LIN {X 0.083,Y -526.031,Z 1290.638,A 0.000,B 0.000,C 90.000,E1 330.745} C_DIS
LIN {X 0.274,Y -522.669,Z 1290.634,A 0.000,B 0.000,C 90.000,E1 329.999} C_DIS
LIN {X 0.174,Y -519.078,Z 1290.630,A 0.000,B 0.000,C 90.000,E1 329.282} C_DIS
LIN {X -0.136,Y -515.219,Z 1290.625,A 0.000,B 0.000,C 90.000,E1 328.584} C_DIS
LIN {X 0.084,Y -506.189,Z 1290.616,A 0.000,B 0.000,C 90.000,E1 326.786} C_DIS
LIN {X -0.322,Y -502.917,Z 1290.611,A 0.000,B 0.000,C 90.000,E1 326.087} C_DIS
LIN {X 0.061,Y -500.954,Z 1290.608,A 0.000,B 0.000,C 90.000,E1 325.468} C_DIS
LIN {X -0.178,Y -499.307,Z 1290.605,A 0.000,B 0.000,C 90.000,E1 324.895} C_DIS
LIN {X -0.148,Y -497.632,Z 1290.600,A 0.000,B 0.000,C 90.000,E1 323.989} C_DIS
LIN {X 0.154,Y -496.578,Z 1290.595,A 0.000,B 0.000,C 90.000,E1 323.050} C_DIS
LIN {X 0.309,Y -495.797,Z 1290.588,A 0.000,B 0.000,C 90.000,E1 321.823} C_DIS
LIN {X -0.218,Y -495.460,Z 1290.578,A 0.000,B 0.000,C 90.000,E1 320.070} C_DIS
LIN {X -0.116,Y -495.714,Z 1290.568,A 0.000,B 0.000,C 90.000,E1 318.243} C_DIS
LIN {X -0.048,Y -495.867,Z 1290.561,A 0.000,B 0.000,C 90.000,E1 317.025} C_DIS
LIN {X 0.028,Y -496.080,Z 1290.551,A 0.000,B 0.000,C 90.000,E1 315.202} C_DIS
LIN {X 0.109,Y -496.318,Z 1290.541,A 0.000,B 0.000,C 90.000,E1 313.380} C_DIS
LIN {X -0.001,Y -496.479,Z 1290.536,A 0.000,B 0.000,C 90.000,E1 312.486} C_DIS
LIN {X -0.140,Y -496.309,Z 1290.531,A 0.000,B 0.000,C 90.000,E1 311.595} C_DIS
LIN {X -0.099,Y -495.936,Z 1290.528,A 0.000,B 0.000,C 90.000,E1 310.987} C_DIS
LIN {X -0.062,Y -495.305,Z 1290.524,A 0.000,B 0.000,C 90.000,E1 310.378} C_DIS
LIN {X -0.031,Y -494.227,Z 1290.521,A 0.000,B 0.000,C 90.000,E1 309.769} C_DIS
LIN {X -0.175,Y -493.450,Z 1290.519,A 0.000,B 0.000,C 90.000,E1 309.483} C_DIS
LIN {X 0.062,Y -492.278,Z 1290.518,A 0.000,B 0.000,C 90.000,E1 309.152} C_DIS
LIN {X 0.225,Y -490.280,Z 1290.516,A 0.000,B 0.000,C 90.000,E1 308.830} C_DIS
LIN {X 0.189,Y -473.095,Z 1290.501,A 0.000,B 0.000,C 90.000,E1 306.217} C_DIS
LIN {X -0.156,Y -457.653,Z 1290.486,A 0.000,B 0.000,C 90.000,E1 303.579} C_DIS
LIN {X 0.164,Y -443.847,Z 1290.471,A 0.000,B 0.000,C 90.000,E1 300.797} C_DIS
LIN {X 0.057,Y -430.915,Z 1290.455,A 0.000,B 0.000,C 90.000,E1 297.847} C_DIS
LIN {X -0.181,Y -420.207,Z 1290.439,A 0.000,B 0.000,C 90.000,E1 295.027} C_DIS
LIN {X -0.114,Y -410.389,Z 1290.422,A 0.000,B 0.000,C 90.000,E1 291.950} C_DIS
LIN {X 0.091,Y -403.056,Z 1290.407,A 0.000,B 0.000,C 90.000,E1 289.214} C_DIS
LIN {X 0.053,Y -403.058,Z 1290.407,A 0.000,B 0.000,C 90.000,E1 289.214} C_DIS
LIN {X -0.122,Y -404.702,Z 1290.395,A 0.000,B 0.000,C 90.000,E1 287.094} C_DIS
LIN {X -0.130,Y -406.128,Z 1290.364,A 0.000,B 0.000,C 90.000,E1 281.535} C_DIS
LIN {X -0.087,Y -405.724,Z 1290.356,A 0.000,B 0.000,C 90.000,E1 280.141} C_DIS
LIN {X -0.037,Y -405.688,Z 1290.333,A 0.000,B 0.000,C 90.000,E1 275.967} C_DIS
LIN {X 0.000,Y -403.466,Z 1290.304,A 0.000,B 0.000,C 90.000,E1 270.745} C_DIS
LIN {X -0.032,Y -403.253,Z 1290.302,A 0.000,B 0.000,C 90.000,E1 270.401} C_DIS
LIN {X 0.147,Y -398.874,Z 1290.271,A 0.000,B 0.000,C 90.000,E1 264.780} C_DIS
LIN {X 0.045,Y -393.348,Z 1290.244,A 0.000,B 0.000,C 90.000,E1 259.859} C_DIS
LIN {X -0.033,Y -392.777,Z 1290.240,A 0.000,B 0.000,C 90.000,E1 259.162} C_DIS
LIN {X 0.116,Y -390.126,Z 1290.230,A 0.000,B 0.000,C 90.000,E1 257.465} C_DIS
LIN {X 0.079,Y -390.127,Z 1290.230,A 0.000,B 0.000,C 90.000,E1 257.465} C_DIS
LIN {X -0.160,Y -397.492,Z 1290.208,A 0.000,B 0.000,C 90.000,E1 253.504} C_DIS
LIN {X -0.205,Y -405.860,Z 1290.189,A 0.000,B 0.000,C 90.000,E1 250.007} C_DIS
LIN {X 0.003,Y -414.932,Z 1290.172,A 0.000,B 0.000,C 90.000,E1 246.869} C_DIS
LIN {X 0.012,Y -426.168,Z 1290.154,A 0.000,B 0.000,C 90.000,E1 243.640} C_DIS
LIN {X -0.200,Y -438.462,Z 1290.137,A 0.000,B 0.000,C 90.000,E1 240.667} C_DIS
LIN {X -0.039,Y -451.639,Z 1290.121,A 0.000,B 0.000,C 90.000,E1 237.867} C_DIS
LIN {X 0.118,Y -455.806,Z 1290.117,A 0.000,B 0.000,C 90.000,E1 237.041} C_DIS
LIN {X -0.149,Y -456.438,Z 1290.116,A 0.000,B 0.000,C 90.000,E1 236.914} C_DIS
LIN {X -0.045,Y -457.275,Z 1290.114,A 0.000,B 0.000,C 90.000,E1 236.580} C_DIS
LIN {X 0.059,Y -457.846,Z 1290.113,A 0.000,B 0.000,C 90.000,E1 236.246} C_DIS
LIN {X 0.155,Y -458.486,Z 1290.109,A 0.000,B 0.000,C 90.000,E1 235.595} C_DIS
LIN {X -0.001,Y -458.776,Z 1290.105,A 0.000,B 0.000,C 90.000,E1 234.975} C_DIS
LIN {X 0.222,Y -458.863,Z 1290.100,A 0.000,B 0.000,C 90.000,E1 233.989} C_DIS
LIN {X 0.076,Y -458.567,Z 1290.095,A 0.000,B 0.000,C 90.000,E1 233.050} C_DIS
LIN {X -0.223,Y -457.721,Z 1290.084,A 0.000,B 0.000,C 90.000,E1 231.170} C_DIS
LIN {X 0.129,Y -456.793,Z 1290.070,A 0.000,B 0.000,C 90.000,E1 228.566} C_DIS
LIN {X -0.042,Y -456.332,Z 1290.061,A 0.000,B 0.000,C 90.000,E1 226.986} C_DIS
LIN {X -0.130,Y -455.866,Z 1290.047,A 0.000,B 0.000,C 90.000,E1 224.433} C_DIS
LIN {X -0.137,Y -456.231,Z 1290.027,A 0.000,B 0.000,C 90.000,E1 220.906} C_DIS
LIN {X -0.095,Y -457.345,Z 1290.013,A 0.000,B 0.000,C 90.000,E1 218.338} C_DIS
LIN {X 0.015,Y -461.089,Z 1289.985,A 0.000,B 0.000,C 90.000,E1 213.214} C_DIS
LIN {X -0.103,Y -463.575,Z 1289.972,A 0.000,B 0.000,C 90.000,E1 211.003} C_DIS
LIN {X -0.167,Y -467.366,Z 1289.955,A 0.000,B 0.000,C 90.000,E1 207.847} C_DIS
LIN {X 0.254,Y -470.340,Z 1289.942,A 0.000,B 0.000,C 90.000,E1 205.591} C_DIS
LIN {X -0.201,Y -472.677,Z 1289.934,A 0.000,B 0.000,C 90.000,E1 204.079} C_DIS
LIN {X 0.177,Y -476.348,Z 1289.920,A 0.000,B 0.000,C 90.000,E1 201.535} C_DIS
LIN {X -0.111,Y -479.825,Z 1289.908,A 0.000,B 0.000,C 90.000,E1 199.396} C_DIS
LIN {X 0.138,Y -482.883,Z 1289.897,A 0.000,B 0.000,C 90.000,E1 197.511} C_DIS
LIN {X 0.160,Y -485.987,Z 1289.887,A 0.000,B 0.000,C 90.000,E1 195.662} C_DIS
LIN {X 0.129,Y -489.110,Z 1289.877,A 0.000,B 0.000,C 90.000,E1 193.828} C_DIS
LIN {X 0.160,Y -491.727,Z 1289.869,A 0.000,B 0.000,C 90.000,E1 192.299} C_DIS
LIN {X -0.049,Y -495.342,Z 1289.857,A 0.000,B 0.000,C 90.000,E1 190.197} C_DIS
LIN {X -0.171,Y -498.512,Z 1289.847,A 0.000,B 0.000,C 90.000,E1 188.398} C_DIS
LIN {X 0.073,Y -500.049,Z 1289.842,A 0.000,B 0.000,C 90.000,E1 187.466} C_DIS
LIN {X -0.082,Y -503.094,Z 1289.832,A 0.000,B 0.000,C 90.000,E1 185.682} C_DIS
LIN {X -0.090,Y -505.461,Z 1289.823,A 0.000,B 0.000,C 90.000,E1 184.188} C_DIS
LIN {X 0.046,Y -507.381,Z 1289.817,A 0.000,B 0.000,C 90.000,E1 182.980} C_DIS
LIN {X 0.080,Y -509.631,Z 1289.808,A 0.000,B 0.000,C 90.000,E1 181.489} C_DIS
LIN {X 0.148,Y -511.671,Z 1289.800,A 0.000,B 0.000,C 90.000,E1 180.000} C_DIS
LIN {X -0.259,Y -513.528,Z 1289.792,A 0.000,B 0.000,C 90.000,E1 178.568} C_DIS
LIN {X -0.036,Y -514.856,Z 1289.785,A 0.000,B 0.000,C 90.000,E1 177.364} C_DIS
LIN {X -0.232,Y -515.732,Z 1289.781,A 0.000,B 0.000,C 90.000,E1 176.502} C_DIS
LIN {X 0.096,Y -516.454,Z 1289.776,A 0.000,B 0.000,C 90.000,E1 175.584} C_DIS
LIN {X -0.110,Y -517.200,Z 1289.769,A 0.000,B 0.000,C 90.000,E1 174.432} C_DIS
LIN {X 0.191,Y -517.807,Z 1289.761,A 0.000,B 0.000,C 90.000,E1 172.932} C_DIS
LIN {X 0.081,Y -517.978,Z 1289.756,A 0.000,B 0.000,C 90.000,E1 172.064} C_DIS
LIN {X -0.037,Y -517.969,Z 1289.750,A 0.000,B 0.000,C 90.000,E1 170.905} C_DIS
LIN {X -0.160,Y -517.604,Z 1289.743,A 0.000,B 0.000,C 90.000,E1 169.746} C_DIS
LIN {X -0.199,Y -516.890,Z 1289.736,A 0.000,B 0.000,C 90.000,E1 168.578} C_DIS
LIN {X -0.237,Y -516.175,Z 1289.732,A 0.000,B 0.000,C 90.000,E1 167.701} C_DIS
LIN {X -0.204,Y -514.467,Z 1289.723,A 0.000,B 0.000,C 90.000,E1 166.228} C_DIS
LIN {X -0.251,Y -513.714,Z 1289.720,A 0.000,B 0.000,C 90.000,E1 165.644} C_DIS
LIN {X -0.142,Y -511.511,Z 1289.712,A 0.000,B 0.000,C 90.000,E1 164.157} C_DIS
LIN {X 0.020,Y -508.537,Z 1289.702,A 0.000,B 0.000,C 90.000,E1 162.362} C_DIS
LIN {X 0.154,Y -506.908,Z 1289.697,A 0.000,B 0.000,C 90.000,E1 161.456} C_DIS
LIN {X 0.147,Y -503.458,Z 1289.682,A 0.000,B 0.000,C 90.000,E1 158.773} C_DIS
LIN {X -0.069,Y -502.868,Z 1289.677,A 0.000,B 0.000,C 90.000,E1 157.901} C_DIS
LIN {X 0.176,Y -502.812,Z 1289.672,A 0.000,B 0.000,C 90.000,E1 156.975} C_DIS
LIN {X 0.257,Y -502.910,Z 1289.671,A 0.000,B 0.000,C 90.000,E1 156.666} C_DIS
LIN {X -0.125,Y -503.191,Z 1289.669,A 0.000,B 0.000,C 90.000,E1 156.410} C_DIS
LIN {X 0.035,Y -504.310,Z 1289.666,A 0.000,B 0.000,C 90.000,E1 155.793} C_DIS
LIN {X -0.259,Y -506.027,Z 1289.662,A 0.000,B 0.000,C 90.000,E1 155.229} C_DIS
LIN {X -0.162,Y -507.409,Z 1289.661,A 0.000,B 0.000,C 90.000,E1 154.921} C_DIS
LIN {X 0.330,Y -508.042,Z 1289.660,A 0.000,B 0.000,C 90.000,E1 154.717} C_DIS
LIN {X 0.020,Y -512.118,Z 1289.656,A 0.000,B 0.000,C 90.000,E1 154.076} C_DIS
LIN {X 0.060,Y -519.658,Z 1289.650,A 0.000,B 0.000,C 90.000,E1 152.999} C_DIS
LIN {X -0.046,Y -526.944,Z 1289.645,A 0.000,B 0.000,C 90.000,E1 152.153} C_DIS
LIN {X -0.094,Y -532.653,Z 1289.641,A 0.000,B 0.000,C 90.000,E1 151.435} C_DIS
LIN {X 0.050,Y -540.691,Z 1289.637,A 0.000,B 0.000,C 90.000,E1 150.589} C_DIS
LIN {X -0.215,Y -549.206,Z 1289.633,A 0.000,B 0.000,C 90.000,E1 149.871} C_DIS
LIN {X -0.326,Y -559.542,Z 1289.628,A 0.000,B 0.000,C 90.000,E1 149.076} C_DIS
LIN {X 0.230,Y -576.226,Z 1289.620,A 0.000,B 0.000,C 90.000,E1 147.582} C_DIS
LIN {X -0.049,Y -580.302,Z 1289.618,A 0.000,B 0.000,C 90.000,E1 147.248} C_DIS
LIN {X -0.255,Y -589.432,Z 1289.613,A 0.000,B 0.000,C 90.000,E1 146.421} C_DIS
LIN {X 0.108,Y -595.843,Z 1289.610,A 0.000,B 0.000,C 90.000,E1 145.754} C_DIS
LIN {X 0.154,Y -601.955,Z 1289.606,A 0.000,B 0.000,C 90.000,E1 145.102} C_DIS
LIN {X 0.039,Y -609.405,Z 1289.601,A 0.000,B 0.000,C 90.000,E1 144.196} C_DIS
LIN {X -0.255,Y -613.214,Z 1289.598,A 0.000,B 0.000,C 90.000,E1 143.703} C_DIS
LIN {X -0.190,Y -617.440,Z 1289.595,A 0.000,B 0.000,C 90.000,E1 143.050} C_DIS
LIN {X -0.084,Y -621.380,Z 1289.591,A 0.000,B 0.000,C 90.000,E1 142.396} C_DIS
LIN {X 0.031,Y -625.965,Z 1289.587,A 0.000,B 0.000,C 90.000,E1 141.618} C_DIS
LIN {X 0.207,Y -629.372,Z 1289.583,A 0.000,B 0.000,C 90.000,E1 140.964} C_DIS
LIN {X -0.056,Y -631.927,Z 1289.580,A 0.000,B 0.000,C 90.000,E1 140.481} C_DIS
LIN {X 0.037,Y -636.667,Z 1289.575,A 0.000,B 0.000,C 90.000,E1 139.461} C_DIS
LIN {X 0.215,Y -639.855,Z 1289.571,A 0.000,B 0.000,C 90.000,E1 138.690} C_DIS
LIN {X -0.165,Y -644.960,Z 1289.564,A 0.000,B 0.000,C 90.000,E1 137.472} C_DIS
LIN {X -0.091,Y -650.633,Z 1289.555,A 0.000,B 0.000,C 90.000,E1 135.972} C_DIS
LIN {X -0.331,Y -655.263,Z 1289.549,A 0.000,B 0.000,C 90.000,E1 134.757} C_DIS
LIN {X 0.006,Y -658.983,Z 1289.543,A 0.000,B 0.000,C 90.000,E1 133.743} C_DIS
LIN {X -0.119,Y -664.500,Z 1289.535,A 0.000,B 0.000,C 90.000,E1 132.285} C_DIS
LIN {X -0.103,Y -668.044,Z 1289.530,A 0.000,B 0.000,C 90.000,E1 131.310} C_DIS
LIN {X -0.033,Y -671.477,Z 1289.524,A 0.000,B 0.000,C 90.000,E1 130.334} C_DIS
LIN {X 0.093,Y -675.495,Z 1289.517,A 0.000,B 0.000,C 90.000,E1 129.116} C_DIS
LIN {X -0.154,Y -679.235,Z 1289.511,A 0.000,B 0.000,C 90.000,E1 127.935} C_DIS
LIN {X 0.191,Y -682.761,Z 1289.504,A 0.000,B 0.000,C 90.000,E1 126.710} C_DIS
LIN {X -0.030,Y -684.097,Z 1289.501,A 0.000,B 0.000,C 90.000,E1 126.251} C_DIS
LIN {X 0.396,Y -687.135,Z 1289.495,A 0.000,B 0.000,C 90.000,E1 125.025} C_DIS
LIN {X 0.080,Y -689.867,Z 1289.488,A 0.000,B 0.000,C 90.000,E1 123.865} C_DIS
LIN {X -0.049,Y -691.316,Z 1289.484,A 0.000,B 0.000,C 90.000,E1 123.166} C_DIS
LIN {X -0.300,Y -693.492,Z 1289.478,A 0.000,B 0.000,C 90.000,E1 122.005} C_DIS
LIN {X -0.035,Y -696.136,Z 1289.469,A 0.000,B 0.000,C 90.000,E1 120.335} C_DIS
LIN {X -0.321,Y -698.144,Z 1289.461,A 0.000,B 0.000,C 90.000,E1 118.949} C_DIS
LIN {X 0.121,Y -699.124,Z 1289.456,A 0.000,B 0.000,C 90.000,E1 117.975} C_DIS
LIN {X -0.049,Y -699.821,Z 1289.450,A 0.000,B 0.000,C 90.000,E1 117.052} C_DIS
LIN {X 0.092,Y -699.981,Z 1289.445,A 0.000,B 0.000,C 90.000,E1 116.104} C_DIS
LIN {X 0.003,Y -699.865,Z 1289.443,A 0.000,B 0.000,C 90.000,E1 115.643} C_DIS
LIN {X 0.243,Y -699.577,Z 1289.440,A 0.000,B 0.000,C 90.000,E1 115.155} C_DIS
LIN {X -0.147,Y -699.127,Z 1289.437,A 0.000,B 0.000,C 90.000,E1 114.719} C_DIS
LIN {X -0.250,Y -698.336,Z 1289.435,A 0.000,B 0.000,C 90.000,E1 114.259} C_DIS
LIN {X -0.009,Y -696.698,Z 1289.432,A 0.000,B 0.000,C 90.000,E1 113.770} C_DIS
LIN {X 0.249,Y -695.719,Z 1289.431,A 0.000,B 0.000,C 90.000,E1 113.515} C_DIS
LIN {X -0.161,Y -692.441,Z 1289.428,A 0.000,B 0.000,C 90.000,E1 113.078} C_DIS
LIN {X -0.041,Y -691.488,Z 1289.427,A 0.000,B 0.000,C 90.000,E1 112.950} C_DIS
LIN {X 0.079,Y -690.067,Z 1289.427,A 0.000,B 0.000,C 90.000,E1 112.823} C_DIS
LIN {X -0.317,Y -683.445,Z 1289.425,A 0.000,B 0.000,C 90.000,E1 112.461} C_DIS
LIN {X 0.136,Y -681.325,Z 1289.424,A 0.000,B 0.000,C 90.000,E1 112.333} C_DIS
LIN {X -0.044,Y -678.247,Z 1289.424,A 0.000,B 0.000,C 90.000,E1 112.259} C_DIS
LIN {X -0.416,Y -671.472,Z 1289.423,A 0.000,B 0.000,C 90.000,E1 112.153} C_DIS
LIN {X 0.035,Y -668.069,Z 1289.423,A 0.000,B 0.000,C 90.000,E1 112.078} C_DIS
LIN {X 0.350,Y -663.498,Z 1289.423,A 0.000,B 0.000,C 90.000,E1 112.025} C_DIS
LIN {X 0.281,Y -643.375,Z 1289.423,A 0.000,B 0.000,C 90.000,E1 112.025} C_DIS
LIN {X -0.170,Y -641.107,Z 1289.422,A 0.000,B 0.000,C 90.000,E1 112.025} C_DIS
LIN {X -0.112,Y -638.394,Z 1289.422,A 0.000,B 0.000,C 90.000,E1 111.950} C_DIS
LIN {X -0.146,Y -638.300,Z 1289.422,A 0.000,B 0.000,C 90.000,E1 111.950} C_DIS
LIN {X -0.141,Y -639.010,Z 1289.421,A 0.000,B 0.000,C 90.000,E1 111.770} C_DIS
LIN {X -0.153,Y -641.523,Z 1289.419,A 0.000,B 0.000,C 90.000,E1 111.354} C_DIS
LIN {X -0.195,Y -647.571,Z 1289.414,A 0.000,B 0.000,C 90.000,E1 110.556} C_DIS
LIN {X -0.090,Y -650.233,Z 1289.412,A 0.000,B 0.000,C 90.000,E1 110.174} C_DIS
LIN {X -0.339,Y -654.176,Z 1289.409,A 0.000,B 0.000,C 90.000,E1 109.577} C_DIS
LIN {X 0.331,Y -658.195,Z 1289.405,A 0.000,B 0.000,C 90.000,E1 108.779} C_DIS
LIN {X 0.201,Y -661.735,Z 1289.400,A 0.000,B 0.000,C 90.000,E1 108.055} C_DIS
LIN {X 0.101,Y -664.869,Z 1289.396,A 0.000,B 0.000,C 90.000,E1 107.330} C_DIS
LIN {X -0.080,Y -666.764,Z 1289.394,A 0.000,B 0.000,C 90.000,E1 106.858} C_DIS
LIN {X -0.136,Y -669.232,Z 1289.390,A 0.000,B 0.000,C 90.000,E1 106.134} C_DIS
LIN {X -0.284,Y -670.626,Z 1289.387,A 0.000,B 0.000,C 90.000,E1 105.662} C_DIS
LIN {X 0.102,Y -672.899,Z 1289.382,A 0.000,B 0.000,C 90.000,E1 104.662} C_DIS
LIN {X -0.015,Y -673.828,Z 1289.379,A 0.000,B 0.000,C 90.000,E1 104.189} C_DIS
LIN {X 0.034,Y -674.563,Z 1289.376,A 0.000,B 0.000,C 90.000,E1 103.703} C_DIS
LIN {X -0.285,Y -675.371,Z 1289.372,A 0.000,B 0.000,C 90.000,E1 103.008} C_DIS
LIN {X 0.271,Y -675.698,Z 1289.370,A 0.000,B 0.000,C 90.000,E1 102.479} C_DIS
LIN {X 0.169,Y -675.845,Z 1289.367,A 0.000,B 0.000,C 90.000,E1 102.007} C_DIS
LIN {X 0.064,Y -675.815,Z 1289.364,A 0.000,B 0.000,C 90.000,E1 101.535} C_DIS
LIN {X -0.227,Y -675.337,Z 1289.360,A 0.000,B 0.000,C 90.000,E1 100.838} C_DIS
LIN {X 0.324,Y -674.842,Z 1289.357,A 0.000,B 0.000,C 90.000,E1 100.310} C_DIS
LIN {X 0.088,Y -674.132,Z 1289.355,A 0.000,B 0.000,C 90.000,E1 99.849} C_DIS
LIN {X -0.038,Y -673.123,Z 1289.352,A 0.000,B 0.000,C 90.000,E1 99.378} C_DIS
LIN {X -0.281,Y -671.788,Z 1289.349,A 0.000,B 0.000,C 90.000,E1 98.916} C_DIS
LIN {X 0.135,Y -670.122,Z 1289.347,A 0.000,B 0.000,C 90.000,E1 98.398} C_DIS
LIN {X 0.056,Y -669.245,Z 1289.345,A 0.000,B 0.000,C 90.000,E1 98.163} C_DIS
LIN {X -0.205,Y -667.130,Z 1289.343,A 0.000,B 0.000,C 90.000,E1 97.701} C_DIS
LIN {X 0.091,Y -664.060,Z 1289.339,A 0.000,B 0.000,C 90.000,E1 97.068} C_DIS
LIN {X -0.220,Y -660.538,Z 1289.336,A 0.000,B 0.000,C 90.000,E1 96.486} C_DIS
LIN {X 0.116,Y -657.365,Z 1289.333,A 0.000,B 0.000,C 90.000,E1 95.967} C_DIS
LIN {X 0.322,Y -652.937,Z 1289.330,A 0.000,B 0.000,C 90.000,E1 95.334} C_DIS
LIN {X -0.101,Y -649.078,Z 1289.327,A 0.000,B 0.000,C 90.000,E1 94.878} C_DIS
LIN {X 0.155,Y -644.861,Z 1289.324,A 0.000,B 0.000,C 90.000,E1 94.359} C_DIS
LIN {X -0.260,Y -639.140,Z 1289.321,A 0.000,B 0.000,C 90.000,E1 93.784} C_DIS
LIN {X -0.147,Y -633.038,Z 1289.318,A 0.000,B 0.000,C 90.000,E1 93.154} C_DIS
LIN {X 0.159,Y -627.876,Z 1289.315,A 0.000,B 0.000,C 90.000,E1 92.636} C_DIS
LIN {X -0.115,Y -622.794,Z 1289.312,A 0.000,B 0.000,C 90.000,E1 92.178} C_DIS
LIN {X 0.306,Y -615.979,Z 1289.309,A 0.000,B 0.000,C 90.000,E1 91.547} C_DIS
LIN {X -0.011,Y -608.410,Z 1289.306,A 0.000,B 0.000,C 90.000,E1 91.031} C_DIS
LIN {X -0.016,Y -602.179,Z 1289.304,A 0.000,B 0.000,C 90.000,E1 90.630} C_DIS
LIN {X -0.280,Y -595.714,Z 1289.302,A 0.000,B 0.000,C 90.000,E1 90.286} C_DIS
LIN {X -0.162,Y -588.834,Z 1289.300,A 0.000,B 0.000,C 90.000,E1 89.943} C_DIS
LIN {X -0.242,Y -579.881,Z 1289.298,A 0.000,B 0.000,C 90.000,E1 89.599} C_DIS
LIN {X 0.177,Y -576.140,Z 1289.297,A 0.000,B 0.000,C 90.000,E1 89.427} C_DIS
LIN {X -0.083,Y -571.959,Z 1289.296,A 0.000,B 0.000,C 90.000,E1 89.255} C_DIS
LIN {X 0.024,Y -569.925,Z 1289.295,A 0.000,B 0.000,C 90.000,E1 89.026} C_DIS
LIN {X -0.014,Y -569.915,Z 1289.295,A 0.000,B 0.000,C 90.000,E1 89.026} C_DIS
LIN {X -0.276,Y -569.540,Z 1289.294,A 0.000,B 0.000,C 90.000,E1 88.854} C_DIS
LIN {X 0.074,Y -569.423,Z 1289.293,A 0.000,B 0.000,C 90.000,E1 88.682} C_DIS
LIN {X -0.027,Y -569.681,Z 1289.289,A 0.000,B 0.000,C 90.000,E1 87.993} C_DIS
LIN {X -0.222,Y -572.279,Z 1289.272,A 0.000,B 0.000,C 90.000,E1 85.008} C_DIS
LIN {X -0.109,Y -574.690,Z 1289.260,A 0.000,B 0.000,C 90.000,E1 82.818} C_DIS
LIN {X 0.014,Y -576.977,Z 1289.250,A 0.000,B 0.000,C 90.000,E1 80.905} C_DIS
LIN {X 0.205,Y -578.245,Z 1289.244,A 0.000,B 0.000,C 90.000,E1 79.803} C_DIS
LIN {X 0.058,Y -579.558,Z 1289.236,A 0.000,B 0.000,C 90.000,E1 78.465} C_DIS
LIN {X 0.043,Y -580.781,Z 1289.229,A 0.000,B 0.000,C 90.000,E1 77.117} C_DIS
LIN {X 0.186,Y -581.899,Z 1289.221,A 0.000,B 0.000,C 90.000,E1 75.755} C_DIS
LIN {X -0.029,Y -582.693,Z 1289.215,A 0.000,B 0.000,C 90.000,E1 74.700} C_DIS
LIN {X 0.076,Y -583.456,Z 1289.209,A 0.000,B 0.000,C 90.000,E1 73.614} C_DIS
LIN {X 0.166,Y -584.861,Z 1289.197,A 0.000,B 0.000,C 90.000,E1 71.456} C_DIS
LIN {X -0.239,Y -585.464,Z 1289.191,A 0.000,B 0.000,C 90.000,E1 70.423} C_DIS
LIN {X 0.195,Y -586.369,Z 1289.182,A 0.000,B 0.000,C 90.000,E1 68.773} C_DIS
LIN {X -0.147,Y -587.681,Z 1289.170,A 0.000,B 0.000,C 90.000,E1 66.666} C_DIS
LIN {X 0.111,Y -588.676,Z 1289.163,A 0.000,B 0.000,C 90.000,E1 65.305} C_DIS
LIN {X -0.128,Y -590.074,Z 1289.153,A 0.000,B 0.000,C 90.000,E1 63.461} C_DIS
LIN {X 0.139,Y -591.214,Z 1289.145,A 0.000,B 0.000,C 90.000,E1 62.103} C_DIS
LIN {X -0.002,Y -593.003,Z 1289.135,A 0.000,B 0.000,C 90.000,E1 60.255} C_DIS
LIN {X -0.100,Y -594.899,Z 1289.125,A 0.000,B 0.000,C 90.000,E1 58.408} C_DIS
LIN {X -0.034,Y -596.868,Z 1289.114,A 0.000,B 0.000,C 90.000,E1 56.548} C_DIS
LIN {X -0.150,Y -598.434,Z 1289.105,A 0.000,B 0.000,C 90.000,E1 54.975} C_DIS
LIN {X 0.092,Y -599.906,Z 1289.097,A 0.000,B 0.000,C 90.000,E1 53.371} C_DIS
LIN {X 0.010,Y -601.454,Z 1289.086,A 0.000,B 0.000,C 90.000,E1 51.537} C_DIS
LIN {X 0.071,Y -602.250,Z 1289.081,A 0.000,B 0.000,C 90.000,E1 50.481} C_DIS
LIN {X -0.243,Y -602.804,Z 1289.075,A 0.000,B 0.000,C 90.000,E1 49.461} C_DIS
LIN {X -0.370,Y -603.418,Z 1289.067,A 0.000,B 0.000,C 90.000,E1 48.162} C_DIS
LIN {X 0.161,Y -603.881,Z 1289.059,A 0.000,B 0.000,C 90.000,E1 46.539} C_DIS
LIN {X 0.022,Y -604.056,Z 1289.051,A 0.000,B 0.000,C 90.000,E1 45.243} C_DIS
LIN {X -0.112,Y -603.975,Z 1289.044,A 0.000,B 0.000,C 90.000,E1 43.947} C_DIS
LIN {X 0.145,Y -603.764,Z 1289.040,A 0.000,B 0.000,C 90.000,E1 43.137} C_DIS
LIN {X 0.026,Y -603.400,Z 1289.032,A 0.000,B 0.000,C 90.000,E1 41.838} C_DIS
LIN {X -0.136,Y -603.069,Z 1289.028,A 0.000,B 0.000,C 90.000,E1 41.067} C_DIS
LIN {X 0.232,Y -602.241,Z 1289.018,A 0.000,B 0.000,C 90.000,E1 39.197} C_DIS
LIN {X -0.331,Y -601.777,Z 1289.014,A 0.000,B 0.000,C 90.000,E1 38.463} C_DIS
LIN {X 0.077,Y -600.553,Z 1289.006,A 0.000,B 0.000,C 90.000,E1 37.111} C_DIS
LIN {X -0.015,Y -599.026,Z 1288.999,A 0.000,B 0.000,C 90.000,E1 35.804} C_DIS
LIN {X 0.102,Y -597.464,Z 1288.993,A 0.000,B 0.000,C 90.000,E1 34.739} C_DIS
LIN {X -0.371,Y -596.093,Z 1288.989,A 0.000,B 0.000,C 90.000,E1 33.992} C_DIS
LIN {X 0.192,Y -593.975,Z 1288.983,A 0.000,B 0.000,C 90.000,E1 32.880} C_DIS
LIN {X 0.191,Y -592.025,Z 1288.978,A 0.000,B 0.000,C 90.000,E1 32.084} C_DIS
LIN {X -0.327,Y -589.854,Z 1288.974,A 0.000,B 0.000,C 90.000,E1 31.337} C_DIS
LIN {X -0.064,Y -587.336,Z 1288.969,A 0.000,B 0.000,C 90.000,E1 30.512} C_DIS
LIN {X -0.300,Y -585.501,Z 1288.967,A 0.000,B 0.000,C 90.000,E1 30.001} C_DIS
LIN {X 0.253,Y -583.423,Z 1288.964,A 0.000,B 0.000,C 90.000,E1 29.411} C_DIS
LIN {X 0.147,Y -579.877,Z 1288.959,A 0.000,B 0.000,C 90.000,E1 28.615} C_DIS
LIN {X -0.275,Y -575.881,Z 1288.955,A 0.000,B 0.000,C 90.000,E1 27.847} C_DIS
LIN {X 0.039,Y -571.531,Z 1288.950,A 0.000,B 0.000,C 90.000,E1 27.001} C_DIS
LIN {X 0.046,Y -566.470,Z 1288.946,A 0.000,B 0.000,C 90.000,E1 26.181} C_DIS
LIN {X -0.070,Y -562.902,Z 1288.943,A 0.000,B 0.000,C 90.000,E1 25.643} C_DIS
LIN {X -0.054,Y -558.124,Z 1288.939,A 0.000,B 0.000,C 90.000,E1 24.951} C_DIS
LIN {X -0.077,Y -553.050,Z 1288.935,A 0.000,B 0.000,C 90.000,E1 24.259} C_DIS
LIN {X -0.027,Y -548.578,Z 1288.932,A 0.000,B 0.000,C 90.000,E1 23.695} C_DIS
LIN {X 0.102,Y -540.186,Z 1288.926,A 0.000,B 0.000,C 90.000,E1 22.695} C_DIS
LIN {X -0.105,Y -533.983,Z 1288.922,A 0.000,B 0.000,C 90.000,E1 22.025} C_DIS
LIN {X -0.029,Y -524.966,Z 1288.917,A 0.000,B 0.000,C 90.000,E1 21.046} C_DIS
LIN {X -0.119,Y -518.287,Z 1288.913,A 0.000,B 0.000,C 90.000,E1 20.355} C_DIS
LIN {X -0.137,Y -508.782,Z 1288.908,A 0.000,B 0.000,C 90.000,E1 19.396} C_DIS
LIN {X -0.208,Y -503.243,Z 1288.905,A 0.000,B 0.000,C 90.000,E1 18.852} C_DIS
LIN {X 0.077,Y -494.971,Z 1288.900,A 0.000,B 0.000,C 90.000,E1 18.000} C_DIS
LIN {X 0.183,Y -484.832,Z 1288.895,A 0.000,B 0.000,C 90.000,E1 17.040} C_DIS
LIN {X -0.018,Y -474.573,Z 1288.890,A 0.000,B 0.000,C 90.000,E1 16.134} C_DIS
LIN {X 0.122,Y -464.230,Z 1288.885,A 0.000,B 0.000,C 90.000,E1 15.190} C_DIS
LIN {X 0.153,Y -445.086,Z 1288.875,A 0.000,B 0.000,C 90.000,E1 13.411} C_DIS
LIN {X -0.172,Y -424.752,Z 1288.863,A 0.000,B 0.000,C 90.000,E1 11.422} C_DIS
LIN {X 0.099,Y -410.388,Z 1288.855,A 0.000,B 0.000,C 90.000,E1 9.849} C_DIS
LIN {X -0.008,Y -400.468,Z 1288.849,A 0.000,B 0.000,C 90.000,E1 8.746} C_DIS
LIN {X -0.102,Y -396.120,Z 1288.845,A 0.000,B 0.000,C 90.000,E1 8.163} C_DIS
LIN {X 0.035,Y -395.163,Z 1288.844,A 0.000,B 0.000,C 90.000,E1 7.936} C_DIS
LIN {X -0.002,Y -395.150,Z 1288.844,A 0.000,B 0.000,C 90.000,E1 7.936} C_DIS
LIN {X -0.040,Y -395.154,Z 1288.844,A 0.000,B 0.000,C 90.000,E1 7.936} C_DIS
LIN {X -0.078,Y -395.167,Z 1288.844,A 0.000,B 0.000,C 90.000,E1 7.936} C_DIS
LIN {X 0.011,Y -396.219,Z 1288.843,A 0.000,B 0.000,C 90.000,E1 7.757} C_DIS
LIN {X 0.107,Y -399.293,Z 1288.842,A 0.000,B 0.000,C 90.000,E1 7.473} C_DIS
LIN {X -0.156,Y -405.364,Z 1288.839,A 0.000,B 0.000,C 90.000,E1 7.125} C_DIS
LIN {X 0.185,Y -410.605,Z 1288.838,A 0.000,B 0.000,C 90.000,E1 6.777} C_DIS
LIN {X 0.170,Y -416.965,Z 1288.836,A 0.000,B 0.000,C 90.000,E1 6.372} C_DIS
LIN {X -0.097,Y -423.351,Z 1288.833,A 0.000,B 0.000,C 90.000,E1 5.967} C_DIS
LIN {X 0.216,Y -431.048,Z 1288.830,A 0.000,B 0.000,C 90.000,E1 5.334} C_DIS
LIN {X 0.134,Y -441.954,Z 1288.825,A 0.000,B 0.000,C 90.000,E1 4.473} C_DIS
LIN {X 0.220,Y -452.449,Z 1288.820,A 0.000,B 0.000,C 90.000,E1 3.555} C_DIS
LIN {X -0.073,Y -459.789,Z 1288.816,A 0.000,B 0.000,C 90.000,E1 2.922} C_DIS
LIN {X -0.038,Y -466.686,Z 1288.813,A 0.000,B 0.000,C 90.000,E1 2.236} C_DIS
LIN {X 0.051,Y -473.467,Z 1288.808,A 0.000,B 0.000,C 90.000,E1 1.489} C_DIS
LIN {X -0.124,Y -479.927,Z 1288.804,A 0.000,B 0.000,C 90.000,E1 0.745} C_DIS
LIN {X -0.178,Y -483.660,Z 1288.802,A 0.000,B 0.000,C 90.000,E1 0.286} C_DIS
LIN {X 0.011,Y -489.433,Z 1288.797,A 0.000,B 0.000,C 90.000,E1 359.484} C_DIS
LIN {X -0.141,Y -494.604,Z 1288.793,A 0.000,B 0.000,C 90.000,E1 358.740} C_DIS
LIN {X -0.051,Y -500.266,Z 1288.788,A 0.000,B 0.000,C 90.000,E1 357.822} C_DIS
LIN {X -0.110,Y -504.696,Z 1288.784,A 0.000,B 0.000,C 90.000,E1 357.078} C_DIS
LIN {X 0.201,Y -508.065,Z 1288.780,A 0.000,B 0.000,C 90.000,E1 356.445} C_DIS
LIN {X 0.245,Y -511.946,Z 1288.776,A 0.000,B 0.000,C 90.000,E1 355.698} C_DIS
LIN {X 0.242,Y -517.047,Z 1288.771,A 0.000,B 0.000,C 90.000,E1 354.666} C_DIS
LIN {X -0.168,Y -521.582,Z 1288.765,A 0.000,B 0.000,C 90.000,E1 353.685} C_DIS
LIN {X 0.055,Y -524.615,Z 1288.761,A 0.000,B 0.000,C 90.000,E1 352.932} C_DIS
LIN {X 0.004,Y -526.826,Z 1288.758,A 0.000,B 0.000,C 90.000,E1 352.356} C_DIS
LIN {X 0.018,Y -530.883,Z 1288.751,A 0.000,B 0.000,C 90.000,E1 351.197} C_DIS
LIN {X 0.046,Y -533.605,Z 1288.746,A 0.000,B 0.000,C 90.000,E1 350.330} C_DIS
LIN {X 0.192,Y -536.124,Z 1288.742,A 0.000,B 0.000,C 90.000,E1 349.454} C_DIS
LIN {X -0.158,Y -538.320,Z 1288.737,A 0.000,B 0.000,C 90.000,E1 348.634} C_DIS
LIN {X 0.044,Y -540.358,Z 1288.732,A 0.000,B 0.000,C 90.000,E1 347.757} C_DIS
LIN {X -0.184,Y -542.773,Z 1288.726,A 0.000,B 0.000,C 90.000,E1 346.645} C_DIS
LIN {X 0.189,Y -544.323,Z 1288.721,A 0.000,B 0.000,C 90.000,E1 345.755} C_DIS
LIN {X -0.085,Y -545.663,Z 1288.716,A 0.000,B 0.000,C 90.000,E1 344.936} C_DIS
LIN {X 0.032,Y -547.070,Z 1288.710,A 0.000,B 0.000,C 90.000,E1 343.795} C_DIS
LIN {X 0.264,Y -548.264,Z 1288.702,A 0.000,B 0.000,C 90.000,E1 342.362} C_DIS
LIN {X 0.165,Y -548.687,Z 1288.698,A 0.000,B 0.000,C 90.000,E1 341.529} C_DIS
LIN {X -0.277,Y -548.795,Z 1288.693,A 0.000,B 0.000,C 90.000,E1 340.732} C_DIS
LIN {X 0.066,Y -548.428,Z 1288.687,A 0.000,B 0.000,C 90.000,E1 339.571} C_DIS
LIN {X -0.119,Y -548.045,Z 1288.683,A 0.000,B 0.000,C 90.000,E1 339.028} C_DIS
LIN {X -0.099,Y -546.792,Z 1288.677,A 0.000,B 0.000,C 90.000,E1 337.901} C_DIS
LIN {X -0.300,Y -545.907,Z 1288.674,A 0.000,B 0.000,C 90.000,E1 337.358} C_DIS
LIN {X 0.195,Y -544.099,Z 1288.668,A 0.000,B 0.000,C 90.000,E1 336.177} C_DIS
LIN {X -0.059,Y -543.358,Z 1288.666,A 0.000,B 0.000,C 90.000,E1 335.921} C_DIS
LIN {X 0.181,Y -542.845,Z 1288.665,A 0.000,B 0.000,C 90.000,E1 335.613} C_DIS
LIN {X 0.125,Y -539.908,Z 1288.658,A 0.000,B 0.000,C 90.000,E1 334.485} C_DIS
LIN {X 0.045,Y -537.391,Z 1288.654,A 0.000,B 0.000,C 90.000,E1 333.640} C_DIS
LIN {X 0.143,Y -533.647,Z 1288.647,A 0.000,B 0.000,C 90.000,E1 332.487} C_DIS
LIN {X 0.296,Y -531.650,Z 1288.644,A 0.000,B 0.000,C 90.000,E1 331.897} C_DIS
LIN {X -0.285,Y -529.516,Z 1288.641,A 0.000,B 0.000,C 90.000,E1 331.385} C_DIS
LIN {X -0.055,Y -526.481,Z 1288.637,A 0.000,B 0.000,C 90.000,E1 330.639} C_DIS
LIN {X 0.020,Y -521.568,Z 1288.631,A 0.000,B 0.000,C 90.000,E1 329.616} C_DIS
LIN {X 0.174,Y -517.769,Z 1288.627,A 0.000,B 0.000,C 90.000,E1 328.869} C_DIS
LIN {X 0.012,Y -508.458,Z 1288.617,A 0.000,B 0.000,C 90.000,E1 327.120} C_DIS
LIN {X -0.058,Y -503.575,Z 1288.612,A 0.000,B 0.000,C 90.000,E1 326.087} C_DIS
LIN {X 0.015,Y -500.604,Z 1288.607,A 0.000,B 0.000,C 90.000,E1 325.182} C_DIS
LIN {X 0.182,Y -499.198,Z 1288.603,A 0.000,B 0.000,C 90.000,E1 324.562} C_DIS
LIN {X -0.198,Y -497.680,Z 1288.598,A 0.000,B 0.000,C 90.000,E1 323.703} C_DIS
LIN {X 0.106,Y -496.795,Z 1288.593,A 0.000,B 0.000,C 90.000,E1 322.763} C_DIS
LIN {X 0.264,Y -496.105,Z 1288.587,A 0.000,B 0.000,C 90.000,E1 321.537} C_DIS
LIN {X -0.118,Y -495.919,Z 1288.578,A 0.000,B 0.000,C 90.000,E1 320.070} C_DIS
LIN {X -0.005,Y -496.149,Z 1288.568,A 0.000,B 0.000,C 90.000,E1 318.243} C_DIS
LIN {X -0.104,Y -496.360,Z 1288.560,A 0.000,B 0.000,C 90.000,E1 316.743} C_DIS
LIN {X -0.006,Y -496.573,Z 1288.550,A 0.000,B 0.000,C 90.000,E1 314.919} C_DIS
LIN {X -0.225,Y -496.987,Z 1288.536,A 0.000,B 0.000,C 90.000,E1 312.528} C_DIS
LIN {X -0.133,Y -497.179,Z 1288.529,A 0.000,B 0.000,C 90.000,E1 311.310} C_DIS
LIN {X 0.100,Y -496.918,Z 1288.524,A 0.000,B 0.000,C 90.000,E1 310.378} C_DIS
LIN {X 0.006,Y -496.164,Z 1288.519,A 0.000,B 0.000,C 90.000,E1 309.483} C_DIS
LIN {X -0.271,Y -495.267,Z 1288.516,A 0.000,B 0.000,C 90.000,E1 308.910} C_DIS
LIN {X -0.100,Y -494.647,Z 1288.514,A 0.000,B 0.000,C 90.000,E1 308.588} C_DIS
LIN {X 0.147,Y -493.807,Z 1288.513,A 0.000,B 0.000,C 90.000,E1 308.257} C_DIS
LIN {X 0.228,Y -493.242,Z 1288.512,A 0.000,B 0.000,C 90.000,E1 308.096} C_DIS
LIN {X 0.006,Y -492.494,Z 1288.511,A 0.000,B 0.000,C 90.000,E1 307.971} C_DIS
LIN {X -0.187,Y -474.919,Z 1288.496,A 0.000,B 0.000,C 90.000,E1 305.231} C_DIS
LIN {X -0.079,Y -460.039,Z 1288.481,A 0.000,B 0.000,C 90.000,E1 302.546} C_DIS
LIN {X -0.182,Y -446.015,Z 1288.465,A 0.000,B 0.000,C 90.000,E1 299.667} C_DIS
LIN {X -0.019,Y -433.673,Z 1288.448,A 0.000,B 0.000,C 90.000,E1 296.693} C_DIS
LIN {X 0.016,Y -422.378,Z 1288.431,A 0.000,B 0.000,C 90.000,E1 293.515} C_DIS
LIN {X -0.017,Y -412.304,Z 1288.412,A 0.000,B 0.000,C 90.000,E1 290.120} C_DIS
LIN {X -0.181,Y -404.756,Z 1288.395,A 0.000,B 0.000,C 90.000,E1 287.040} C_DIS
LIN {X -0.219,Y -404.745,Z 1288.395,A 0.000,B 0.000,C 90.000,E1 287.040} C_DIS
LIN {X -0.174,Y -406.154,Z 1288.364,A 0.000,B 0.000,C 90.000,E1 281.478} C_DIS
LIN {X -0.075,Y -405.681,Z 1288.333,A 0.000,B 0.000,C 90.000,E1 275.910} C_DIS
LIN {X -0.004,Y -403.567,Z 1288.306,A 0.000,B 0.000,C 90.000,E1 271.031} C_DIS
LIN {X -0.069,Y -403.188,Z 1288.302,A 0.000,B 0.000,C 90.000,E1 270.344} C_DIS
LIN {X 0.165,Y -399.069,Z 1288.273,A 0.000,B 0.000,C 90.000,E1 265.065} C_DIS
LIN {X 0.105,Y -398.785,Z 1288.271,A 0.000,B 0.000,C 90.000,E1 264.723} C_DIS
LIN {X -0.133,Y -393.373,Z 1288.244,A 0.000,B 0.000,C 90.000,E1 259.916} C_DIS
LIN {X 0.215,Y -393.371,Z 1288.244,A 0.000,B 0.000,C 90.000,E1 259.859} C_DIS
LIN {X -0.047,Y -400.123,Z 1288.220,A 0.000,B 0.000,C 90.000,E1 255.574} C_DIS
LIN {X -0.231,Y -408.324,Z 1288.199,A 0.000,B 0.000,C 90.000,E1 251.764} C_DIS
LIN {X 0.067,Y -417.618,Z 1288.179,A 0.000,B 0.000,C 90.000,E1 248.284} C_DIS
LIN {X -0.183,Y -428.146,Z 1288.162,A 0.000,B 0.000,C 90.000,E1 245.101} C_DIS
LIN {X -0.145,Y -439.718,Z 1288.145,A 0.000,B 0.000,C 90.000,E1 242.103} C_DIS
LIN {X 0.180,Y -452.936,Z 1288.129,A 0.000,B 0.000,C 90.000,E1 239.125} C_DIS
LIN {X 0.111,Y -456.914,Z 1288.124,A 0.000,B 0.000,C 90.000,E1 238.329} C_DIS
LIN {X 0.219,Y -458.091,Z 1288.122,A 0.000,B 0.000,C 90.000,E1 237.995} C_DIS
LIN {X -0.058,Y -458.768,Z 1288.121,A 0.000,B 0.000,C 90.000,E1 237.709} C_DIS
LIN {X 0.175,Y -459.535,Z 1288.117,A 0.000,B 0.000,C 90.000,E1 237.041} C_DIS
LIN {X 0.029,Y -459.957,Z 1288.114,A 0.000,B 0.000,C 90.000,E1 236.421} C_DIS
LIN {X -0.114,Y -460.117,Z 1288.110,A 0.000,B 0.000,C 90.000,E1 235.801} C_DIS
LIN {X 0.127,Y -459.954,Z 1288.105,A 0.000,B 0.000,C 90.000,E1 234.815} C_DIS
LIN {X 0.107,Y -459.392,Z 1288.098,A 0.000,B 0.000,C 90.000,E1 233.543} C_DIS
LIN {X -0.074,Y -458.348,Z 1288.085,A 0.000,B 0.000,C 90.000,E1 231.331} C_DIS
LIN {X -0.050,Y -457.412,Z 1288.071,A 0.000,B 0.000,C 90.000,E1 228.771} C_DIS
LIN {X -0.121,Y -456.766,Z 1288.058,A 0.000,B 0.000,C 90.000,E1 226.539} C_DIS
LIN {X 0.173,Y -456.335,Z 1288.041,A 0.000,B 0.000,C 90.000,E1 223.299} C_DIS
LIN {X -0.077,Y -457.117,Z 1288.021,A 0.000,B 0.000,C 90.000,E1 219.806} C_DIS
LIN {X -0.113,Y -457.987,Z 1288.010,A 0.000,B 0.000,C 90.000,E1 217.890} C_DIS
LIN {X 0.018,Y -462.599,Z 1287.979,A 0.000,B 0.000,C 90.000,E1 212.133} C_DIS
LIN {X 0.062,Y -464.415,Z 1287.970,A 0.000,B 0.000,C 90.000,E1 210.541} C_DIS
LIN {X -0.196,Y -467.072,Z 1287.958,A 0.000,B 0.000,C 90.000,E1 208.359} C_DIS
LIN {X 0.216,Y -469.988,Z 1287.945,A 0.000,B 0.000,C 90.000,E1 206.104} C_DIS
LIN {X -0.131,Y -473.184,Z 1287.933,A 0.000,B 0.000,C 90.000,E1 203.951} C_DIS
LIN {X -0.182,Y -476.875,Z 1287.919,A 0.000,B 0.000,C 90.000,E1 201.461} C_DIS
LIN {X -0.003,Y -479.865,Z 1287.909,A 0.000,B 0.000,C 90.000,E1 199.577} C_DIS
LIN {X 0.248,Y -482.968,Z 1287.899,A 0.000,B 0.000,C 90.000,E1 197.692} C_DIS
LIN {X -0.193,Y -486.113,Z 1287.888,A 0.000,B 0.000,C 90.000,E1 195.898} C_DIS
LIN {X -0.106,Y -488.233,Z 1287.881,A 0.000,B 0.000,C 90.000,E1 194.662} C_DIS
LIN {X 0.025,Y -490.871,Z 1287.873,A 0.000,B 0.000,C 90.000,E1 193.119} C_DIS
LIN {X 0.085,Y -492.982,Z 1287.866,A 0.000,B 0.000,C 90.000,E1 191.895} C_DIS
LIN {X 0.182,Y -495.627,Z 1287.858,A 0.000,B 0.000,C 90.000,E1 190.366} C_DIS
LIN {X 0.062,Y -498.844,Z 1287.848,A 0.000,B 0.000,C 90.000,E1 188.568} C_DIS
LIN {X 0.241,Y -500.472,Z 1287.843,A 0.000,B 0.000,C 90.000,E1 187.644} C_DIS
LIN {X 0.157,Y -503.549,Z 1287.833,A 0.000,B 0.000,C 90.000,E1 185.853} C_DIS
LIN {X 0.154,Y -505.985,Z 1287.824,A 0.000,B 0.000,C 90.000,E1 184.359} C_DIS
LIN {X -0.237,Y -507.991,Z 1287.818,A 0.000,B 0.000,C 90.000,E1 183.212} C_DIS
LIN {X -0.165,Y -510.308,Z 1287.809,A 0.000,B 0.000,C 90.000,E1 181.718} C_DIS
LIN {X -0.004,Y -512.007,Z 1287.803,A 0.000,B 0.000,C 90.000,E1 180.516} C_DIS
LIN {X -0.247,Y -513.289,Z 1287.798,A 0.000,B 0.000,C 90.000,E1 179.656} C_DIS
LIN {X -0.098,Y -515.208,Z 1287.790,A 0.000,B 0.000,C 90.000,E1 178.165} C_DIS
LIN {X 0.132,Y -516.543,Z 1287.783,A 0.000,B 0.000,C 90.000,E1 176.963} C_DIS
LIN {X -0.082,Y -517.687,Z 1287.777,A 0.000,B 0.000,C 90.000,E1 175.812} C_DIS
LIN {X 0.178,Y -518.705,Z 1287.769,A 0.000,B 0.000,C 90.000,E1 174.318} C_DIS
LIN {X 0.002,Y -519.303,Z 1287.762,A 0.000,B 0.000,C 90.000,E1 173.166} C_DIS
LIN {X -0.103,Y -519.613,Z 1287.756,A 0.000,B 0.000,C 90.000,E1 172.008} C_DIS
LIN {X -0.199,Y -519.756,Z 1287.749,A 0.000,B 0.000,C 90.000,E1 170.849} C_DIS
LIN {X 0.217,Y -519.550,Z 1287.744,A 0.000,B 0.000,C 90.000,E1 169.926} C_DIS
LIN {X 0.201,Y -519.045,Z 1287.738,A 0.000,B 0.000,C 90.000,E1 168.757} C_DIS
LIN {X 0.177,Y -518.279,Z 1287.731,A 0.000,B 0.000,C 90.000,E1 167.589} C_DIS
LIN {X 0.267,Y -517.406,Z 1287.726,A 0.000,B 0.000,C 90.000,E1 166.700} C_DIS
LIN {X -0.181,Y -515.769,Z 1287.718,A 0.000,B 0.000,C 90.000,E1 165.283} C_DIS
LIN {X -0.060,Y -513.438,Z 1287.708,A 0.000,B 0.000,C 90.000,E1 163.504} C_DIS
LIN {X 0.082,Y -511.677,Z 1287.702,A 0.000,B 0.000,C 90.000,E1 162.308} C_DIS
LIN {X -0.187,Y -509.660,Z 1287.694,A 0.000,B 0.000,C 90.000,E1 160.859} C_DIS
LIN {X -0.217,Y -508.050,Z 1287.684,A 0.000,B 0.000,C 90.000,E1 159.082} C_DIS
LIN {X 0.088,Y -507.644,Z 1287.679,A 0.000,B 0.000,C 90.000,E1 158.156} C_DIS
LIN {X -0.082,Y -507.875,Z 1287.674,A 0.000,B 0.000,C 90.000,E1 157.283} C_DIS
LIN {X 0.118,Y -508.359,Z 1287.671,A 0.000,B 0.000,C 90.000,E1 156.666} C_DIS
LIN {X -0.146,Y -509.257,Z 1287.667,A 0.000,B 0.000,C 90.000,E1 156.102} C_DIS
LIN {X 0.059,Y -510.468,Z 1287.664,A 0.000,B 0.000,C 90.000,E1 155.485} C_DIS
LIN {X -0.196,Y -512.710,Z 1287.661,A 0.000,B 0.000,C 90.000,E1 154.921} C_DIS
LIN {X 0.310,Y -513.608,Z 1287.660,A 0.000,B 0.000,C 90.000,E1 154.717} C_DIS
LIN {X 0.251,Y -515.631,Z 1287.657,A 0.000,B 0.000,C 90.000,E1 154.280} C_DIS
LIN {X -0.159,Y -522.656,Z 1287.651,A 0.000,B 0.000,C 90.000,E1 153.256} C_DIS
LIN {X 0.014,Y -527.329,Z 1287.648,A 0.000,B 0.000,C 90.000,E1 152.666} C_DIS
LIN {X 0.195,Y -529.511,Z 1287.647,A 0.000,B 0.000,C 90.000,E1 152.410} C_DIS
LIN {X 0.037,Y -536.879,Z 1287.642,A 0.000,B 0.000,C 90.000,E1 151.591} C_DIS
LIN {X 0.264,Y -543.431,Z 1287.639,A 0.000,B 0.000,C 90.000,E1 150.923} C_DIS
LIN {X -0.169,Y -547.634,Z 1287.637,A 0.000,B 0.000,C 90.000,E1 150.589} C_DIS
LIN {X -0.207,Y -550.541,Z 1287.635,A 0.000,B 0.000,C 90.000,E1 150.333} C_DIS
LIN {X -0.049,Y -555.841,Z 1287.633,A 0.000,B 0.000,C 90.000,E1 149.871} C_DIS
LIN {X -0.186,Y -562.846,Z 1287.629,A 0.000,B 0.000,C 90.000,E1 149.282} C_DIS
LIN {X 0.105,Y -575.235,Z 1287.623,A 0.000,B 0.000,C 90.000,E1 148.152} C_DIS
LIN {X -0.278,Y -583.311,Z 1287.619,A 0.000,B 0.000,C 90.000,E1 147.454} C_DIS
LIN {X 0.133,Y -589.782,Z 1287.616,A 0.000,B 0.000,C 90.000,E1 146.786} C_DIS
LIN {X -0.042,Y -594.851,Z 1287.613,A 0.000,B 0.000,C 90.000,E1 146.294} C_DIS
LIN {X 0.139,Y -599.657,Z 1287.610,A 0.000,B 0.000,C 90.000,E1 145.754} C_DIS
LIN {X 0.004,Y -603.033,Z 1287.608,A 0.000,B 0.000,C 90.000,E1 145.388} C_DIS
LIN {X 0.167,Y -607.235,Z 1287.605,A 0.000,B 0.000,C 90.000,E1 144.848} C_DIS
LIN {X -0.141,Y -611.242,Z 1287.602,A 0.000,B 0.000,C 90.000,E1 144.356} C_DIS
LIN {X -0.390,Y -614.058,Z 1287.600,A 0.000,B 0.000,C 90.000,E1 143.989} C_DIS
LIN {X 0.175,Y -618.286,Z 1287.596,A 0.000,B 0.000,C 90.000,E1 143.290} C_DIS
LIN {X -0.208,Y -622.205,Z 1287.593,A 0.000,B 0.000,C 90.000,E1 142.683} C_DIS
LIN {X -0.084,Y -626.540,Z 1287.588,A 0.000,B 0.000,C 90.000,E1 141.904} C_DIS
LIN {X 0.077,Y -630.573,Z 1287.584,A 0.000,B 0.000,C 90.000,E1 141.126} C_DIS
LIN {X -0.200,Y -633.642,Z 1287.581,A 0.000,B 0.000,C 90.000,E1 140.517} C_DIS
LIN {X 0.318,Y -638.213,Z 1287.575,A 0.000,B 0.000,C 90.000,E1 139.461} C_DIS
LIN {X 0.088,Y -641.293,Z 1287.571,A 0.000,B 0.000,C 90.000,E1 138.728} C_DIS
LIN {X 0.230,Y -645.212,Z 1287.565,A 0.000,B 0.000,C 90.000,E1 137.715} C_DIS
LIN {X -0.104,Y -649.838,Z 1287.558,A 0.000,B 0.000,C 90.000,E1 136.500} C_DIS
LIN {X 0.073,Y -655.267,Z 1287.550,A 0.000,B 0.000,C 90.000,E1 135.000} C_DIS
LIN {X -0.142,Y -661.516,Z 1287.541,A 0.000,B 0.000,C 90.000,E1 133.299} C_DIS
LIN {X -0.181,Y -666.002,Z 1287.534,A 0.000,B 0.000,C 90.000,E1 132.081} C_DIS
LIN {X -0.137,Y -670.234,Z 1287.527,A 0.000,B 0.000,C 90.000,E1 130.862} C_DIS
LIN {X -0.028,Y -674.269,Z 1287.520,A 0.000,B 0.000,C 90.000,E1 129.644} C_DIS
LIN {X 0.117,Y -677.343,Z 1287.515,A 0.000,B 0.000,C 90.000,E1 128.669} C_DIS
LIN {X -0.124,Y -680.256,Z 1287.510,A 0.000,B 0.000,C 90.000,E1 127.729} C_DIS
LIN {X 0.241,Y -683.689,Z 1287.503,A 0.000,B 0.000,C 90.000,E1 126.503} C_DIS
LIN {X 0.258,Y -686.723,Z 1287.496,A 0.000,B 0.000,C 90.000,E1 125.311} C_DIS
LIN {X -0.268,Y -689.014,Z 1287.491,A 0.000,B 0.000,C 90.000,E1 124.405} C_DIS
LIN {X 0.188,Y -691.128,Z 1287.486,A 0.000,B 0.000,C 90.000,E1 123.420} C_DIS
LIN {X 0.159,Y -693.753,Z 1287.478,A 0.000,B 0.000,C 90.000,E1 122.005} C_DIS
LIN {X 0.182,Y -696.038,Z 1287.470,A 0.000,B 0.000,C 90.000,E1 120.590} C_DIS
LIN {X 0.334,Y -697.124,Z 1287.466,A 0.000,B 0.000,C 90.000,E1 119.873} C_DIS
LIN {X -0.197,Y -698.724,Z 1287.460,A 0.000,B 0.000,C 90.000,E1 118.743} C_DIS
LIN {X -0.019,Y -699.476,Z 1287.456,A 0.000,B 0.000,C 90.000,E1 118.025} C_DIS
LIN {X 0.116,Y -700.223,Z 1287.451,A 0.000,B 0.000,C 90.000,E1 117.078} C_DIS
LIN {X -0.047,Y -700.397,Z 1287.445,A 0.000,B 0.000,C 90.000,E1 116.155} C_DIS
LIN {X -0.083,Y -700.420,Z 1287.444,A 0.000,B 0.000,C 90.000,E1 115.924} C_DIS
LIN {X 0.102,Y -700.045,Z 1287.440,A 0.000,B 0.000,C 90.000,E1 115.207} C_DIS
LIN {X -0.287,Y -699.623,Z 1287.438,A 0.000,B 0.000,C 90.000,E1 114.771} C_DIS
LIN {X 0.248,Y -698.850,Z 1287.435,A 0.000,B 0.000,C 90.000,E1 114.259} C_DIS
LIN {X 0.228,Y -698.208,Z 1287.434,A 0.000,B 0.000,C 90.000,E1 114.027} C_DIS
LIN {X 0.114,Y -696.446,Z 1287.431,A 0.000,B 0.000,C 90.000,E1 113.567} C_DIS
LIN {X -0.036,Y -695.748,Z 1287.430,A 0.000,B 0.000,C 90.000,E1 113.462} C_DIS
LIN {X -0.174,Y -692.349,Z 1287.428,A 0.000,B 0.000,C 90.000,E1 113.003} C_DIS
LIN {X -0.321,Y -691.177,Z 1287.427,A 0.000,B 0.000,C 90.000,E1 112.898} C_DIS
LIN {X -0.200,Y -689.354,Z 1287.427,A 0.000,B 0.000,C 90.000,E1 112.770} C_DIS
LIN {X -0.081,Y -687.123,Z 1287.426,A 0.000,B 0.000,C 90.000,E1 112.642} C_DIS
LIN {X 0.041,Y -683.361,Z 1287.425,A 0.000,B 0.000,C 90.000,E1 112.408} C_DIS
LIN {X -0.134,Y -681.095,Z 1287.424,A 0.000,B 0.000,C 90.000,E1 112.333} C_DIS
LIN {X -0.286,Y -678.946,Z 1287.424,A 0.000,B 0.000,C 90.000,E1 112.280} C_DIS
LIN {X 0.058,Y -670.940,Z 1287.423,A 0.000,B 0.000,C 90.000,E1 112.099} C_DIS
LIN {X -0.234,Y -663.585,Z 1287.423,A 0.000,B 0.000,C 90.000,E1 112.078} C_DIS
LIN {X 0.326,Y -642.480,Z 1287.423,A 0.000,B 0.000,C 90.000,E1 112.025} C_DIS
LIN {X 0.210,Y -639.088,Z 1287.422,A 0.000,B 0.000,C 90.000,E1 111.972} C_DIS
LIN {X -0.208,Y -637.906,Z 1287.422,A 0.000,B 0.000,C 90.000,E1 111.972} C_DIS
LIN {X -0.011,Y -637.823,Z 1287.422,A 0.000,B 0.000,C 90.000,E1 111.950} C_DIS
LIN {X 0.156,Y -638.311,Z 1287.421,A 0.000,B 0.000,C 90.000,E1 111.791} C_DIS
LIN {X 0.180,Y -638.945,Z 1287.421,A 0.000,B 0.000,C 90.000,E1 111.663} C_DIS
LIN {X 0.202,Y -641.377,Z 1287.418,A 0.000,B 0.000,C 90.000,E1 111.280} C_DIS
LIN {X -0.089,Y -647.007,Z 1287.414,A 0.000,B 0.000,C 90.000,E1 110.556} C_DIS
LIN {X 0.014,Y -649.703,Z 1287.412,A 0.000,B 0.000,C 90.000,E1 110.174} C_DIS
LIN {X -0.197,Y -654.347,Z 1287.408,A 0.000,B 0.000,C 90.000,E1 109.450} C_DIS
LIN {X -0.196,Y -657.677,Z 1287.405,A 0.000,B 0.000,C 90.000,E1 108.833} C_DIS
LIN {X 0.291,Y -661.205,Z 1287.401,A 0.000,B 0.000,C 90.000,E1 108.055} C_DIS
LIN {X 0.187,Y -664.386,Z 1287.396,A 0.000,B 0.000,C 90.000,E1 107.330} C_DIS
LIN {X 0.003,Y -666.307,Z 1287.394,A 0.000,B 0.000,C 90.000,E1 106.858} C_DIS
LIN {X -0.057,Y -668.795,Z 1287.390,A 0.000,B 0.000,C 90.000,E1 106.134} C_DIS
LIN {X -0.209,Y -670.241,Z 1287.387,A 0.000,B 0.000,C 90.000,E1 105.662} C_DIS
LIN {X 0.173,Y -672.511,Z 1287.382,A 0.000,B 0.000,C 90.000,E1 104.662} C_DIS
LIN {X 0.054,Y -673.466,Z 1287.379,A 0.000,B 0.000,C 90.000,E1 104.189} C_DIS
LIN {X 0.100,Y -674.230,Z 1287.376,A 0.000,B 0.000,C 90.000,E1 103.703} C_DIS
LIN {X -0.223,Y -675.008,Z 1287.372,A 0.000,B 0.000,C 90.000,E1 103.008} C_DIS
LIN {X -0.328,Y -675.362,Z 1287.370,A 0.000,B 0.000,C 90.000,E1 102.535} C_DIS
LIN {X 0.228,Y -675.508,Z 1287.367,A 0.000,B 0.000,C 90.000,E1 102.007} C_DIS
LIN {X 0.121,Y -675.477,Z 1287.364,A 0.000,B 0.000,C 90.000,E1 101.535} C_DIS
LIN {X -0.173,Y -674.968,Z 1287.360,A 0.000,B 0.000,C 90.000,E1 100.838} C_DIS
LIN {X -0.288,Y -674.471,Z 1287.358,A 0.000,B 0.000,C 90.000,E1 100.366} C_DIS
LIN {X 0.137,Y -673.728,Z 1287.355,A 0.000,B 0.000,C 90.000,E1 99.849} C_DIS
LIN {X 0.008,Y -672.751,Z 1287.352,A 0.000,B 0.000,C 90.000,E1 99.378} C_DIS
LIN {X -0.237,Y -671.414,Z 1287.349,A 0.000,B 0.000,C 90.000,E1 98.916} C_DIS
LIN {X 0.176,Y -669.739,Z 1287.347,A 0.000,B 0.000,C 90.000,E1 98.398} C_DIS
LIN {X 0.096,Y -668.836,Z 1287.345,A 0.000,B 0.000,C 90.000,E1 98.163} C_DIS
LIN {X -0.168,Y -666.721,Z 1287.343,A 0.000,B 0.000,C 90.000,E1 97.701} C_DIS
LIN {X 0.124,Y -663.649,Z 1287.339,A 0.000,B 0.000,C 90.000,E1 97.068} C_DIS
LIN {X -0.191,Y -660.109,Z 1287.336,A 0.000,B 0.000,C 90.000,E1 96.486} C_DIS
LIN {X 0.142,Y -656.886,Z 1287.333,A 0.000,B 0.000,C 90.000,E1 95.967} C_DIS
LIN {X 0.344,Y -652.411,Z 1287.330,A 0.000,B 0.000,C 90.000,E1 95.334} C_DIS
LIN {X -0.082,Y -648.526,Z 1287.327,A 0.000,B 0.000,C 90.000,E1 94.878} C_DIS
LIN {X 0.170,Y -644.245,Z 1287.324,A 0.000,B 0.000,C 90.000,E1 94.359} C_DIS
LIN {X 0.266,Y -638.376,Z 1287.321,A 0.000,B 0.000,C 90.000,E1 93.726} C_DIS
LIN {X -0.152,Y -633.491,Z 1287.318,A 0.000,B 0.000,C 90.000,E1 93.269} C_DIS
LIN {X 0.190,Y -628.344,Z 1287.315,A 0.000,B 0.000,C 90.000,E1 92.751} C_DIS
LIN {X 0.251,Y -622.151,Z 1287.312,A 0.000,B 0.000,C 90.000,E1 92.178} C_DIS
LIN {X 0.287,Y -615.431,Z 1287.309,A 0.000,B 0.000,C 90.000,E1 91.604} C_DIS
LIN {X -0.092,Y -609.468,Z 1287.307,A 0.000,B 0.000,C 90.000,E1 91.203} C_DIS
LIN {X -0.242,Y -603.182,Z 1287.304,A 0.000,B 0.000,C 90.000,E1 90.802} C_DIS
LIN {X 0.281,Y -595.102,Z 1287.302,A 0.000,B 0.000,C 90.000,E1 90.286} C_DIS
LIN {X 0.039,Y -589.975,Z 1287.300,A 0.000,B 0.000,C 90.000,E1 90.057} C_DIS
LIN {X -0.054,Y -582.828,Z 1287.299,A 0.000,B 0.000,C 90.000,E1 89.771} C_DIS
LIN {X 0.157,Y -575.815,Z 1287.297,A 0.000,B 0.000,C 90.000,E1 89.484} C_DIS
LIN {X 0.190,Y -572.195,Z 1287.296,A 0.000,B 0.000,C 90.000,E1 89.312} C_DIS
LIN {X 0.141,Y -572.097,Z 1287.296,A 0.000,B 0.000,C 90.000,E1 89.312} C_DIS
LIN {X 0.239,Y -569.807,Z 1287.295,A 0.000,B 0.000,C 90.000,E1 89.026} C_DIS
LIN {X 0.197,Y -569.781,Z 1287.295,A 0.000,B 0.000,C 90.000,E1 89.026} C_DIS
LIN {X -0.047,Y -569.409,Z 1287.294,A 0.000,B 0.000,C 90.000,E1 88.854} C_DIS
LIN {X -0.074,Y -569.368,Z 1287.292,A 0.000,B 0.000,C 90.000,E1 88.568} C_DIS
LIN {X 0.126,Y -572.483,Z 1287.271,A 0.000,B 0.000,C 90.000,E1 84.723} C_DIS
LIN {X 0.234,Y -574.908,Z 1287.259,A 0.000,B 0.000,C 90.000,E1 82.534} C_DIS
LIN {X -0.218,Y -577.189,Z 1287.248,A 0.000,B 0.000,C 90.000,E1 80.679} C_DIS
LIN {X 0.073,Y -578.395,Z 1287.242,A 0.000,B 0.000,C 90.000,E1 79.567} C_DIS
LIN {X -0.071,Y -579.668,Z 1287.235,A 0.000,B 0.000,C 90.000,E1 78.229} C_DIS
LIN {X 0.259,Y -580.651,Z 1287.229,A 0.000,B 0.000,C 90.000,E1 77.117} C_DIS
LIN {X -0.164,Y -581.771,Z 1287.221,A 0.000,B 0.000,C 90.000,E1 75.811} C_DIS
LIN {X 0.183,Y -582.569,Z 1287.215,A 0.000,B 0.000,C 90.000,E1 74.700} C_DIS
LIN {X -0.047,Y -583.467,Z 1287.208,A 0.000,B 0.000,C 90.000,E1 73.378} C_DIS
LIN {X 0.039,Y -584.928,Z 1287.196,A 0.000,B 0.000,C 90.000,E1 71.221} C_DIS
LIN {X -0.019,Y -586.054,Z 1287.184,A 0.000,B 0.000,C 90.000,E1 69.082} C_DIS
LIN {X 0.171,Y -587.356,Z 1287.172,A 0.000,B 0.000,C 90.000,E1 66.922} C_DIS
LIN {X -0.227,Y -588.521,Z 1287.163,A 0.000,B 0.000,C 90.000,E1 65.357} C_DIS
LIN {X 0.173,Y -589.740,Z 1287.154,A 0.000,B 0.000,C 90.000,E1 63.717} C_DIS
LIN {X -0.192,Y -591.091,Z 1287.145,A 0.000,B 0.000,C 90.000,E1 62.153} C_DIS
LIN {X 0.186,Y -592.882,Z 1287.135,A 0.000,B 0.000,C 90.000,E1 60.255} C_DIS
LIN {X 0.086,Y -594.778,Z 1287.125,A 0.000,B 0.000,C 90.000,E1 58.408} C_DIS
LIN {X 0.151,Y -596.746,Z 1287.114,A 0.000,B 0.000,C 90.000,E1 56.548} C_DIS
LIN {X 0.031,Y -598.297,Z 1287.105,A 0.000,B 0.000,C 90.000,E1 54.975} C_DIS
LIN {X -0.210,Y -599.768,Z 1287.097,A 0.000,B 0.000,C 90.000,E1 53.417} C_DIS
LIN {X -0.060,Y -601.112,Z 1287.088,A 0.000,B 0.000,C 90.000,E1 51.823} C_DIS
LIN {X -0.137,Y -602.103,Z 1287.081,A 0.000,B 0.000,C 90.000,E1 50.517} C_DIS
LIN {X 0.177,Y -602.792,Z 1287.073,A 0.000,B 0.000,C 90.000,E1 49.175} C_DIS
LIN {X 0.045,Y -603.373,Z 1287.066,A 0.000,B 0.000,C 90.000,E1 47.877} C_DIS
LIN {X -0.109,Y -603.756,Z 1287.059,A 0.000,B 0.000,C 90.000,E1 46.581} C_DIS
LIN {X -0.036,Y -603.925,Z 1287.053,A 0.000,B 0.000,C 90.000,E1 45.526} C_DIS
LIN {X 0.251,Y -603.890,Z 1287.046,A 0.000,B 0.000,C 90.000,E1 44.190} C_DIS
LIN {X 0.093,Y -603.750,Z 1287.041,A 0.000,B 0.000,C 90.000,E1 43.419} C_DIS
LIN {X 0.188,Y -603.295,Z 1287.033,A 0.000,B 0.000,C 90.000,E1 41.838} C_DIS
LIN {X 0.025,Y -602.964,Z 1287.028,A 0.000,B 0.000,C 90.000,E1 41.067} C_DIS
LIN {X 0.389,Y -602.137,Z 1287.018,A 0.000,B 0.000,C 90.000,E1 39.197} C_DIS
LIN {X -0.175,Y -601.675,Z 1287.014,A 0.000,B 0.000,C 90.000,E1 38.463} C_DIS
LIN {X -0.247,Y -600.446,Z 1287.006,A 0.000,B 0.000,C 90.000,E1 37.156} C_DIS
LIN {X 0.137,Y -598.904,Z 1286.999,A 0.000,B 0.000,C 90.000,E1 35.804} C_DIS
LIN {X 0.018,Y -597.771,Z 1286.995,A 0.000,B 0.000,C 90.000,E1 35.025} C_DIS
LIN {X -0.115,Y -596.494,Z 1286.990,A 0.000,B 0.000,C 90.000,E1 34.246} C_DIS
LIN {X 0.122,Y -594.457,Z 1286.984,A 0.000,B 0.000,C 90.000,E1 33.166} C_DIS
LIN {X -0.374,Y -592.631,Z 1286.980,A 0.000,B 0.000,C 90.000,E1 32.418} C_DIS
LIN {X -0.072,Y -590.501,Z 1286.976,A 0.000,B 0.000,C 90.000,E1 31.592} C_DIS
LIN {X 0.009,Y -588.949,Z 1286.973,A 0.000,B 0.000,C 90.000,E1 31.052} C_DIS
LIN {X -0.039,Y -586.304,Z 1286.968,A 0.000,B 0.000,C 90.000,E1 30.256} C_DIS
LIN {X -0.279,Y -584.382,Z 1286.965,A 0.000,B 0.000,C 90.000,E1 29.745} C_DIS
LIN {X -0.242,Y -582.212,Z 1286.962,A 0.000,B 0.000,C 90.000,E1 29.205} C_DIS
LIN {X 0.216,Y -579.139,Z 1286.958,A 0.000,B 0.000,C 90.000,E1 28.487} C_DIS
LIN {X -0.213,Y -575.090,Z 1286.954,A 0.000,B 0.000,C 90.000,E1 27.719} C_DIS
LIN {X 0.173,Y -571.449,Z 1286.950,A 0.000,B 0.000,C 90.000,E1 27.001} C_DIS
LIN {X 0.178,Y -566.385,Z 1286.946,A 0.000,B 0.000,C 90.000,E1 26.181} C_DIS
LIN {X -0.091,Y -563.711,Z 1286.943,A 0.000,B 0.000,C 90.000,E1 25.796} C_DIS
LIN {X 0.177,Y -558.990,Z 1286.939,A 0.000,B 0.000,C 90.000,E1 25.079} C_DIS
LIN {X 0.050,Y -552.952,Z 1286.935,A 0.000,B 0.000,C 90.000,E1 24.259} C_DIS
LIN {X 0.098,Y -548.474,Z 1286.932,A 0.000,B 0.000,C 90.000,E1 23.695} C_DIS
LIN {X 0.015,Y -540.088,Z 1286.926,A 0.000,B 0.000,C 90.000,E1 22.717} C_DIS
LIN {X -0.015,Y -533.820,Z 1286.922,A 0.000,B 0.000,C 90.000,E1 22.025} C_DIS
LIN {X -0.036,Y -524.711,Z 1286.917,A 0.000,B 0.000,C 90.000,E1 21.046} C_DIS
LIN {X -0.127,Y -518.024,Z 1286.913,A 0.000,B 0.000,C 90.000,E1 20.355} C_DIS
LIN {X -0.259,Y -507.129,Z 1286.907,A 0.000,B 0.000,C 90.000,E1 19.268} C_DIS
LIN {X 0.074,Y -494.684,Z 1286.900,A 0.000,B 0.000,C 90.000,E1 18.000} C_DIS
LIN {X -0.165,Y -486.021,Z 1286.896,A 0.000,B 0.000,C 90.000,E1 17.221} C_DIS
LIN {X 0.104,Y -475.812,Z 1286.891,A 0.000,B 0.000,C 90.000,E1 16.260} C_DIS
LIN {X 0.192,Y -463.954,Z 1286.885,A 0.000,B 0.000,C 90.000,E1 15.190} C_DIS
LIN {X 0.244,Y -444.863,Z 1286.875,A 0.000,B 0.000,C 90.000,E1 13.411} C_DIS
LIN {X -0.107,Y -421.712,Z 1286.862,A 0.000,B 0.000,C 90.000,E1 11.130} C_DIS
LIN {X 0.169,Y -400.374,Z 1286.849,A 0.000,B 0.000,C 90.000,E1 8.746} C_DIS
LIN {X 0.055,Y -396.009,Z 1286.845,A 0.000,B 0.000,C 90.000,E1 8.163} C_DIS
LIN {X -0.005,Y -395.181,Z 1286.844,A 0.000,B 0.000,C 90.000,E1 7.992} C_DIS
LIN {X -0.043,Y -395.159,Z 1286.844,A 0.000,B 0.000,C 90.000,E1 7.992} C_DIS
LIN {X 0.044,Y -395.199,Z 1286.844,A 0.000,B 0.000,C 90.000,E1 7.936} C_DIS
LIN {X 0.006,Y -395.216,Z 1286.844,A 0.000,B 0.000,C 90.000,E1 7.936} C_DIS
LIN {X 0.170,Y -396.173,Z 1286.843,A 0.000,B 0.000,C 90.000,E1 7.757} C_DIS
LIN {X -0.128,Y -399.243,Z 1286.842,A 0.000,B 0.000,C 90.000,E1 7.530} C_DIS
LIN {X -0.074,Y -403.575,Z 1286.840,A 0.000,B 0.000,C 90.000,E1 7.239} C_DIS
LIN {X -0.025,Y -410.511,Z 1286.838,A 0.000,B 0.000,C 90.000,E1 6.834} C_DIS
LIN {X -0.040,Y -416.873,Z 1286.836,A 0.000,B 0.000,C 90.000,E1 6.429} C_DIS
LIN {X 0.082,Y -423.251,Z 1286.833,A 0.000,B 0.000,C 90.000,E1 5.967} C_DIS
LIN {X -0.022,Y -430.944,Z 1286.830,A 0.000,B 0.000,C 90.000,E1 5.391} C_DIS
LIN {X 0.032,Y -441.672,Z 1286.825,A 0.000,B 0.000,C 90.000,E1 4.531} C_DIS
LIN {X 0.183,Y -452.171,Z 1286.820,A 0.000,B 0.000,C 90.000,E1 3.612} C_DIS
LIN {X -0.070,Y -459.506,Z 1286.817,A 0.000,B 0.000,C 90.000,E1 2.980} C_DIS
LIN {X -0.041,Y -466.472,Z 1286.813,A 0.000,B 0.000,C 90.000,E1 2.293} C_DIS
LIN {X 0.062,Y -473.294,Z 1286.809,A 0.000,B 0.000,C 90.000,E1 1.547} C_DIS
LIN {X -0.218,Y -479.510,Z 1286.805,A 0.000,B 0.000,C 90.000,E1 0.859} C_DIS
LIN {X -0.091,Y -484.435,Z 1286.801,A 0.000,B 0.000,C 90.000,E1 0.229} C_DIS
LIN {X 0.013,Y -489.872,Z 1286.797,A 0.000,B 0.000,C 90.000,E1 359.484} C_DIS
LIN {X -0.136,Y -495.044,Z 1286.793,A 0.000,B 0.000,C 90.000,E1 358.740} C_DIS
LIN {X -0.040,Y -500.739,Z 1286.788,A 0.000,B 0.000,C 90.000,E1 357.822} C_DIS
LIN {X -0.095,Y -505.201,Z 1286.784,A 0.000,B 0.000,C 90.000,E1 357.078} C_DIS
LIN {X -0.084,Y -509.376,Z 1286.780,A 0.000,B 0.000,C 90.000,E1 356.331} C_DIS
LIN {X -0.033,Y -513.223,Z 1286.776,A 0.000,B 0.000,C 90.000,E1 355.584} C_DIS
LIN {X 0.027,Y -518.293,Z 1286.770,A 0.000,B 0.000,C 90.000,E1 354.546} C_DIS
LIN {X 0.097,Y -522.738,Z 1286.764,A 0.000,B 0.000,C 90.000,E1 353.514} C_DIS
LIN {X 0.041,Y -526.331,Z 1286.759,A 0.000,B 0.000,C 90.000,E1 352.648} C_DIS
LIN {X 0.044,Y -530.469,Z 1286.753,A 0.000,B 0.000,C 90.000,E1 351.489} C_DIS
LIN {X 0.066,Y -533.339,Z 1286.748,A 0.000,B 0.000,C 90.000,E1 350.622} C_DIS
LIN {X 0.207,Y -535.904,Z 1286.743,A 0.000,B 0.000,C 90.000,E1 349.746} C_DIS
LIN {X -0.146,Y -538.196,Z 1286.738,A 0.000,B 0.000,C 90.000,E1 348.926} C_DIS
LIN {X 0.128,Y -540.947,Z 1286.732,A 0.000,B 0.000,C 90.000,E1 347.757} C_DIS
LIN {X -0.091,Y -543.361,Z 1286.726,A 0.000,B 0.000,C 90.000,E1 346.645} C_DIS
LIN {X 0.072,Y -544.474,Z 1286.723,A 0.000,B 0.000,C 90.000,E1 346.061} C_DIS
LIN {X 0.022,Y -546.334,Z 1286.716,A 0.000,B 0.000,C 90.000,E1 344.936} C_DIS
LIN {X 0.147,Y -547.737,Z 1286.710,A 0.000,B 0.000,C 90.000,E1 343.795} C_DIS
LIN {X 0.052,Y -548.492,Z 1286.705,A 0.000,B 0.000,C 90.000,E1 342.960} C_DIS
LIN {X -0.042,Y -549.173,Z 1286.701,A 0.000,B 0.000,C 90.000,E1 342.127} C_DIS
LIN {X 0.041,Y -549.537,Z 1286.696,A 0.000,B 0.000,C 90.000,E1 341.275} C_DIS
LIN {X -0.133,Y -549.600,Z 1286.693,A 0.000,B 0.000,C 90.000,E1 340.732} C_DIS
LIN {X -0.042,Y -549.377,Z 1286.688,A 0.000,B 0.000,C 90.000,E1 339.880} C_DIS
LIN {X -0.221,Y -549.132,Z 1286.685,A 0.000,B 0.000,C 90.000,E1 339.337} C_DIS
LIN {X 0.059,Y -548.341,Z 1286.680,A 0.000,B 0.000,C 90.000,E1 338.465} C_DIS
LIN {X 0.128,Y -547.304,Z 1286.676,A 0.000,B 0.000,C 90.000,E1 337.614} C_DIS
LIN {X -0.110,Y -544.979,Z 1286.668,A 0.000,B 0.000,C 90.000,E1 336.230} C_DIS
LIN {X -0.114,Y -543.906,Z 1286.665,A 0.000,B 0.000,C 90.000,E1 335.665} C_DIS
LIN {X 0.128,Y -543.271,Z 1286.663,A 0.000,B 0.000,C 90.000,E1 335.357} C_DIS
LIN {X -0.127,Y -542.376,Z 1286.662,A 0.000,B 0.000,C 90.000,E1 335.101} C_DIS
LIN {X -0.107,Y -541.056,Z 1286.659,A 0.000,B 0.000,C 90.000,E1 334.537} C_DIS
LIN {X -0.170,Y -538.591,Z 1286.654,A 0.000,B 0.000,C 90.000,E1 333.691} C_DIS
LIN {X -0.048,Y -534.826,Z 1286.647,A 0.000,B 0.000,C 90.000,E1 332.538} C_DIS
LIN {X 0.012,Y -530.608,Z 1286.641,A 0.000,B 0.000,C 90.000,E1 331.385} C_DIS
LIN {X -0.008,Y -527.621,Z 1286.637,A 0.000,B 0.000,C 90.000,E1 330.667} C_DIS
LIN {X -0.115,Y -522.605,Z 1286.631,A 0.000,B 0.000,C 90.000,E1 329.665} C_DIS
LIN {X -0.049,Y -519.581,Z 1286.628,A 0.000,B 0.000,C 90.000,E1 329.076} C_DIS
LIN {X 0.257,Y -507.846,Z 1286.616,A 0.000,B 0.000,C 90.000,E1 326.834} C_DIS
LIN {X -0.134,Y -504.344,Z 1286.612,A 0.000,B 0.000,C 90.000,E1 326.135} C_DIS
LIN {X -0.222,Y -501.237,Z 1286.607,A 0.000,B 0.000,C 90.000,E1 325.261} C_DIS
LIN {X 0.240,Y -499.788,Z 1286.604,A 0.000,B 0.000,C 90.000,E1 324.609} C_DIS
LIN {X 0.272,Y -498.212,Z 1286.599,A 0.000,B 0.000,C 90.000,E1 323.703} C_DIS
LIN {X 0.015,Y -497.481,Z 1286.595,A 0.000,B 0.000,C 90.000,E1 323.130} C_DIS
LIN {X 0.183,Y -496.687,Z 1286.589,A 0.000,B 0.000,C 90.000,E1 321.904} C_DIS
LIN {X -0.188,Y -496.306,Z 1286.580,A 0.000,B 0.000,C 90.000,E1 320.436} C_DIS
LIN {X -0.063,Y -496.548,Z 1286.570,A 0.000,B 0.000,C 90.000,E1 318.609} C_DIS
LIN {X 0.063,Y -496.806,Z 1286.560,A 0.000,B 0.000,C 90.000,E1 316.782} C_DIS
LIN {X -0.192,Y -497.032,Z 1286.550,A 0.000,B 0.000,C 90.000,E1 315.000} C_DIS
LIN {X 0.306,Y -497.430,Z 1286.536,A 0.000,B 0.000,C 90.000,E1 312.528} C_DIS
LIN {X -0.107,Y -497.757,Z 1286.528,A 0.000,B 0.000,C 90.000,E1 311.067} C_DIS
LIN {X -0.056,Y -497.842,Z 1286.525,A 0.000,B 0.000,C 90.000,E1 310.458} C_DIS
LIN {X -0.140,Y -497.644,Z 1286.520,A 0.000,B 0.000,C 90.000,E1 309.564} C_DIS
LIN {X 0.161,Y -497.038,Z 1286.515,A 0.000,B 0.000,C 90.000,E1 308.624} C_DIS
LIN {X 0.202,Y -496.334,Z 1286.511,A 0.000,B 0.000,C 90.000,E1 308.016} C_DIS
LIN {X 0.066,Y -495.853,Z 1286.510,A 0.000,B 0.000,C 90.000,E1 307.729} C_DIS
LIN {X -0.069,Y -495.241,Z 1286.508,A 0.000,B 0.000,C 90.000,E1 307.443} C_DIS
LIN {X -0.207,Y -494.392,Z 1286.506,A 0.000,B 0.000,C 90.000,E1 307.156} C_DIS
LIN {X -0.127,Y -493.836,Z 1286.505,A 0.000,B 0.000,C 90.000,E1 306.996} C_DIS
LIN {X 0.050,Y -493.107,Z 1286.505,A 0.000,B 0.000,C 90.000,E1 306.824} C_DIS
LIN {X -0.005,Y -476.240,Z 1286.489,A 0.000,B 0.000,C 90.000,E1 304.072} C_DIS
LIN {X -0.100,Y -461.185,Z 1286.474,A 0.000,B 0.000,C 90.000,E1 301.258} C_DIS
LIN {X 0.004,Y -447.852,Z 1286.458,A 0.000,B 0.000,C 90.000,E1 298.359} C_DIS
LIN {X 0.036,Y -436.149,Z 1286.441,A 0.000,B 0.000,C 90.000,E1 295.412} C_DIS
LIN {X 0.121,Y -426.000,Z 1286.425,A 0.000,B 0.000,C 90.000,E1 292.408} C_DIS
LIN {X 0.097,Y -416.449,Z 1286.406,A 0.000,B 0.000,C 90.000,E1 289.033} C_DIS
LIN {X 0.208,Y -407.944,Z 1286.385,A 0.000,B 0.000,C 90.000,E1 285.245} C_DIS
LIN {X -0.125,Y -405.115,Z 1286.376,A 0.000,B 0.000,C 90.000,E1 283.772} C_DIS
LIN {X -0.163,Y -405.116,Z 1286.376,A 0.000,B 0.000,C 90.000,E1 283.772} C_DIS
LIN {X -0.136,Y -406.152,Z 1286.364,A 0.000,B 0.000,C 90.000,E1 281.478} C_DIS
LIN {X -0.038,Y -405.682,Z 1286.333,A 0.000,B 0.000,C 90.000,E1 275.910} C_DIS
LIN {X 0.034,Y -403.568,Z 1286.306,A 0.000,B 0.000,C 90.000,E1 271.031} C_DIS
LIN {X -0.031,Y -403.194,Z 1286.302,A 0.000,B 0.000,C 90.000,E1 270.344} C_DIS
LIN {X 0.201,Y -399.072,Z 1286.273,A 0.000,B 0.000,C 90.000,E1 265.065} C_DIS
LIN {X 0.143,Y -398.792,Z 1286.271,A 0.000,B 0.000,C 90.000,E1 264.723} C_DIS
LIN {X 0.110,Y -396.575,Z 1286.262,A 0.000,B 0.000,C 90.000,E1 263.053} C_DIS
LIN {X 0.071,Y -396.573,Z 1286.261,A 0.000,B 0.000,C 90.000,E1 263.053} C_DIS
LIN {X 0.144,Y -402.593,Z 1286.234,A 0.000,B 0.000,C 90.000,E1 258.049} C_DIS
LIN {X -0.141,Y -410.228,Z 1286.211,A 0.000,B 0.000,C 90.000,E1 253.921} C_DIS
LIN {X -0.048,Y -418.451,Z 1286.192,A 0.000,B 0.000,C 90.000,E1 250.477} C_DIS
LIN {X -0.102,Y -428.442,Z 1286.173,A 0.000,B 0.000,C 90.000,E1 247.102} C_DIS
LIN {X -0.139,Y -439.651,Z 1286.155,A 0.000,B 0.000,C 90.000,E1 243.948} C_DIS
LIN {X -0.076,Y -451.888,Z 1286.139,A 0.000,B 0.000,C 90.000,E1 241.001} C_DIS
LIN {X 0.048,Y -458.614,Z 1286.131,A 0.000,B 0.000,C 90.000,E1 239.537} C_DIS
LIN {X 0.163,Y -459.612,Z 1286.129,A 0.000,B 0.000,C 90.000,E1 239.203} C_DIS
LIN {X -0.113,Y -460.209,Z 1286.127,A 0.000,B 0.000,C 90.000,E1 238.918} C_DIS
LIN {X -0.106,Y -460.910,Z 1286.124,A 0.000,B 0.000,C 90.000,E1 238.280} C_DIS
LIN {X -0.247,Y -461.253,Z 1286.120,A 0.000,B 0.000,C 90.000,E1 237.661} C_DIS
LIN {X -0.254,Y -461.332,Z 1286.115,A 0.000,B 0.000,C 90.000,E1 236.707} C_DIS
LIN {X 0.253,Y -461.261,Z 1286.111,A 0.000,B 0.000,C 90.000,E1 236.008} C_DIS
LIN {X -0.015,Y -460.574,Z 1286.104,A 0.000,B 0.000,C 90.000,E1 234.769} C_DIS
LIN {X -0.165,Y -459.446,Z 1286.092,A 0.000,B 0.000,C 90.000,E1 232.557} C_DIS
LIN {X -0.159,Y -458.596,Z 1286.081,A 0.000,B 0.000,C 90.000,E1 230.642} C_DIS
LIN {X 0.121,Y -457.934,Z 1286.071,A 0.000,B 0.000,C 90.000,E1 228.690} C_DIS
LIN {X 0.065,Y -457.271,Z 1286.058,A 0.000,B 0.000,C 90.000,E1 226.458} C_DIS
LIN {X 0.035,Y -456.832,Z 1286.042,A 0.000,B 0.000,C 90.000,E1 223.581} C_DIS
LIN {X -0.225,Y -457.518,Z 1286.023,A 0.000,B 0.000,C 90.000,E1 220.092} C_DIS
LIN {X 0.121,Y -458.393,Z 1286.010,A 0.000,B 0.000,C 90.000,E1 217.810} C_DIS
LIN {X 0.026,Y -462.999,Z 1285.978,A 0.000,B 0.000,C 90.000,E1 212.084} C_DIS
LIN {X -0.082,Y -464.831,Z 1285.969,A 0.000,B 0.000,C 90.000,E1 210.512} C_DIS
LIN {X 0.114,Y -465.994,Z 1285.964,A 0.000,B 0.000,C 90.000,E1 209.539} C_DIS
LIN {X 0.235,Y -469.106,Z 1285.950,A 0.000,B 0.000,C 90.000,E1 207.001} C_DIS
LIN {X 0.068,Y -472.162,Z 1285.938,A 0.000,B 0.000,C 90.000,E1 204.823} C_DIS
LIN {X 0.073,Y -474.499,Z 1285.929,A 0.000,B 0.000,C 90.000,E1 203.259} C_DIS
LIN {X -0.118,Y -478.323,Z 1285.916,A 0.000,B 0.000,C 90.000,E1 200.791} C_DIS
LIN {X 0.090,Y -481.843,Z 1285.903,A 0.000,B 0.000,C 90.000,E1 198.598} C_DIS
LIN {X 0.231,Y -485.045,Z 1285.893,A 0.000,B 0.000,C 90.000,E1 196.732} C_DIS
LIN {X 0.176,Y -488.265,Z 1285.883,A 0.000,B 0.000,C 90.000,E1 194.898} C_DIS
LIN {X -0.167,Y -490.930,Z 1285.874,A 0.000,B 0.000,C 90.000,E1 193.411} C_DIS
LIN {X -0.109,Y -493.607,Z 1285.866,A 0.000,B 0.000,C 90.000,E1 191.883} C_DIS
LIN {X -0.101,Y -496.306,Z 1285.858,A 0.000,B 0.000,C 90.000,E1 190.366} C_DIS
LIN {X -0.208,Y -499.591,Z 1285.848,A 0.000,B 0.000,C 90.000,E1 188.568} C_DIS
LIN {X -0.099,Y -501.750,Z 1285.841,A 0.000,B 0.000,C 90.000,E1 187.352} C_DIS
LIN {X -0.089,Y -504.389,Z 1285.833,A 0.000,B 0.000,C 90.000,E1 185.853} C_DIS
LIN {X -0.077,Y -506.885,Z 1285.824,A 0.000,B 0.000,C 90.000,E1 184.359} C_DIS
LIN {X 0.052,Y -508.935,Z 1285.818,A 0.000,B 0.000,C 90.000,E1 183.154} C_DIS
LIN {X 0.143,Y -511.318,Z 1285.809,A 0.000,B 0.000,C 90.000,E1 181.661} C_DIS
LIN {X 0.165,Y -513.994,Z 1285.800,A 0.000,B 0.000,C 90.000,E1 179.885} C_DIS
LIN {X 0.261,Y -516.382,Z 1285.790,A 0.000,B 0.000,C 90.000,E1 178.108} C_DIS
LIN {X -0.008,Y -517.797,Z 1285.783,A 0.000,B 0.000,C 90.000,E1 176.963} C_DIS
LIN {X -0.203,Y -519.015,Z 1285.777,A 0.000,B 0.000,C 90.000,E1 175.812} C_DIS
LIN {X 0.082,Y -520.149,Z 1285.769,A 0.000,B 0.000,C 90.000,E1 174.318} C_DIS
LIN {X -0.074,Y -520.840,Z 1285.762,A 0.000,B 0.000,C 90.000,E1 173.166} C_DIS
LIN {X -0.231,Y -521.369,Z 1285.754,A 0.000,B 0.000,C 90.000,E1 171.724} C_DIS
LIN {X -0.228,Y -521.510,Z 1285.749,A 0.000,B 0.000,C 90.000,E1 170.849} C_DIS
LIN {X 0.211,Y -521.335,Z 1285.743,A 0.000,B 0.000,C 90.000,E1 169.634} C_DIS
LIN {X 0.220,Y -521.079,Z 1285.738,A 0.000,B 0.000,C 90.000,E1 168.757} C_DIS
LIN {X -0.282,Y -520.195,Z 1285.730,A 0.000,B 0.000,C 90.000,E1 167.353} C_DIS
LIN {X -0.173,Y -519.128,Z 1285.723,A 0.000,B 0.000,C 90.000,E1 166.172} C_DIS
LIN {X -0.068,Y -518.223,Z 1285.718,A 0.000,B 0.000,C 90.000,E1 165.283} C_DIS
LIN {X 0.011,Y -517.023,Z 1285.712,A 0.000,B 0.000,C 90.000,E1 164.102} C_DIS
LIN {X -0.193,Y -514.998,Z 1285.702,A 0.000,B 0.000,C 90.000,E1 162.362} C_DIS
LIN {X 0.135,Y -513.599,Z 1285.695,A 0.000,B 0.000,C 90.000,E1 161.148} C_DIS
LIN {X -0.211,Y -512.646,Z 1285.689,A 0.000,B 0.000,C 90.000,E1 160.007} C_DIS
LIN {X 0.260,Y -512.185,Z 1285.682,A 0.000,B 0.000,C 90.000,E1 158.773} C_DIS
LIN {X -0.055,Y -512.413,Z 1285.677,A 0.000,B 0.000,C 90.000,E1 157.922} C_DIS
LIN {X -0.178,Y -513.106,Z 1285.672,A 0.000,B 0.000,C 90.000,E1 157.050} C_DIS
LIN {X -0.292,Y -514.502,Z 1285.667,A 0.000,B 0.000,C 90.000,E1 156.177} C_DIS
LIN {X 0.165,Y -516.019,Z 1285.664,A 0.000,B 0.000,C 90.000,E1 155.537} C_DIS
LIN {X -0.178,Y -517.017,Z 1285.663,A 0.000,B 0.000,C 90.000,E1 155.281} C_DIS
LIN {X -0.084,Y -520.122,Z 1285.659,A 0.000,B 0.000,C 90.000,E1 154.537} C_DIS
LIN {X 0.119,Y -522.634,Z 1285.656,A 0.000,B 0.000,C 90.000,E1 154.076} C_DIS
LIN {X -0.050,Y -526.483,Z 1285.653,A 0.000,B 0.000,C 90.000,E1 153.512} C_DIS
LIN {X -0.090,Y -532.165,Z 1285.649,A 0.000,B 0.000,C 90.000,E1 152.794} C_DIS
LIN {X -0.065,Y -537.138,Z 1285.646,A 0.000,B 0.000,C 90.000,E1 152.231} C_DIS
LIN {X -0.184,Y -543.645,Z 1285.642,A 0.000,B 0.000,C 90.000,E1 151.563} C_DIS
LIN {X -0.128,Y -549.007,Z 1285.639,A 0.000,B 0.000,C 90.000,E1 151.051} C_DIS
LIN {X 0.015,Y -554.435,Z 1285.636,A 0.000,B 0.000,C 90.000,E1 150.511} C_DIS
LIN {X -0.167,Y -562.822,Z 1285.632,A 0.000,B 0.000,C 90.000,E1 149.793} C_DIS
LIN {X 0.048,Y -577.741,Z 1285.625,A 0.000,B 0.000,C 90.000,E1 148.408} C_DIS
LIN {X -0.047,Y -586.753,Z 1285.620,A 0.000,B 0.000,C 90.000,E1 147.533} C_DIS
LIN {X -0.026,Y -595.655,Z 1285.615,A 0.000,B 0.000,C 90.000,E1 146.628} C_DIS
LIN {X -0.221,Y -601.326,Z 1285.611,A 0.000,B 0.000,C 90.000,E1 146.008} C_DIS
LIN {X -0.022,Y -604.655,Z 1285.609,A 0.000,B 0.000,C 90.000,E1 145.595} C_DIS
LIN {X 0.153,Y -608.748,Z 1285.606,A 0.000,B 0.000,C 90.000,E1 145.055} C_DIS
LIN {X -0.109,Y -611.677,Z 1285.604,A 0.000,B 0.000,C 90.000,E1 144.689} C_DIS
LIN {X 0.144,Y -614.467,Z 1285.602,A 0.000,B 0.000,C 90.000,E1 144.276} C_DIS
LIN {X 0.193,Y -619.397,Z 1285.597,A 0.000,B 0.000,C 90.000,E1 143.497} C_DIS
LIN {X 0.312,Y -623.251,Z 1285.594,A 0.000,B 0.000,C 90.000,E1 142.844} C_DIS
LIN {X 0.106,Y -626.098,Z 1285.591,A 0.000,B 0.000,C 90.000,E1 142.351} C_DIS
LIN {X 0.128,Y -631.341,Z 1285.585,A 0.000,B 0.000,C 90.000,E1 141.331} C_DIS
LIN {X 0.364,Y -633.773,Z 1285.583,A 0.000,B 0.000,C 90.000,E1 140.803} C_DIS
LIN {X -0.112,Y -639.250,Z 1285.575,A 0.000,B 0.000,C 90.000,E1 139.585} C_DIS
LIN {X -0.329,Y -642.238,Z 1285.571,A 0.000,B 0.000,C 90.000,E1 138.852} C_DIS
LIN {X -0.171,Y -646.053,Z 1285.566,A 0.000,B 0.000,C 90.000,E1 137.838} C_DIS
LIN {X 0.044,Y -649.685,Z 1285.560,A 0.000,B 0.000,C 90.000,E1 136.824} C_DIS
LIN {X 0.260,Y -654.094,Z 1285.553,A 0.000,B 0.000,C 90.000,E1 135.567} C_DIS
LIN {X 0.109,Y -657.590,Z 1285.548,A 0.000,B 0.000,C 90.000,E1 134.595} C_DIS
LIN {X -0.040,Y -662.866,Z 1285.540,A 0.000,B 0.000,C 90.000,E1 133.137} C_DIS
LIN {X -0.058,Y -667.206,Z 1285.533,A 0.000,B 0.000,C 90.000,E1 131.919} C_DIS
LIN {X 0.000,Y -670.480,Z 1285.527,A 0.000,B 0.000,C 90.000,E1 130.943} C_DIS
LIN {X 0.105,Y -673.659,Z 1285.522,A 0.000,B 0.000,C 90.000,E1 129.967} C_DIS
LIN {X 0.266,Y -677.495,Z 1285.516,A 0.000,B 0.000,C 90.000,E1 128.749} C_DIS
LIN {X 0.009,Y -679.652,Z 1285.511,A 0.000,B 0.000,C 90.000,E1 128.051} C_DIS
LIN {X -0.170,Y -683.104,Z 1285.505,A 0.000,B 0.000,C 90.000,E1 126.870} C_DIS
LIN {X 0.214,Y -685.632,Z 1285.500,A 0.000,B 0.000,C 90.000,E1 125.884} C_DIS
LIN {X 0.267,Y -688.541,Z 1285.493,A 0.000,B 0.000,C 90.000,E1 124.692} C_DIS
LIN {X -0.236,Y -690.704,Z 1285.488,A 0.000,B 0.000,C 90.000,E1 123.785} C_DIS
LIN {X 0.220,Y -692.124,Z 1285.484,A 0.000,B 0.000,C 90.000,E1 123.038} C_DIS
LIN {X -0.248,Y -693.910,Z 1285.478,A 0.000,B 0.000,C 90.000,E1 122.133} C_DIS
LIN {X 0.125,Y -695.852,Z 1285.472,A 0.000,B 0.000,C 90.000,E1 120.924} C_DIS
LIN {X -0.075,Y -697.350,Z 1285.467,A 0.000,B 0.000,C 90.000,E1 120.001} C_DIS
LIN {X 0.007,Y -698.984,Z 1285.460,A 0.000,B 0.000,C 90.000,E1 118.821} C_DIS
LIN {X -0.157,Y -699.986,Z 1285.455,A 0.000,B 0.000,C 90.000,E1 117.897} C_DIS
LIN {X 0.032,Y -700.556,Z 1285.451,A 0.000,B 0.000,C 90.000,E1 117.180} C_DIS
LIN {X 0.182,Y -700.808,Z 1285.446,A 0.000,B 0.000,C 90.000,E1 116.232} C_DIS
LIN {X -0.206,Y -700.785,Z 1285.443,A 0.000,B 0.000,C 90.000,E1 115.796} C_DIS
LIN {X -0.290,Y -700.582,Z 1285.441,A 0.000,B 0.000,C 90.000,E1 115.335} C_DIS
LIN {X -0.042,Y -700.130,Z 1285.438,A 0.000,B 0.000,C 90.000,E1 114.847} C_DIS
LIN {X 0.131,Y -699.037,Z 1285.434,A 0.000,B 0.000,C 90.000,E1 114.131} C_DIS
LIN {X -0.263,Y -697.314,Z 1285.432,A 0.000,B 0.000,C 90.000,E1 113.695} C_DIS
LIN {X -0.281,Y -696.142,Z 1285.430,A 0.000,B 0.000,C 90.000,E1 113.462} C_DIS
LIN {X 0.224,Y -692.666,Z 1285.428,A 0.000,B 0.000,C 90.000,E1 112.950} C_DIS
LIN {X 0.344,Y -691.465,Z 1285.427,A 0.000,B 0.000,C 90.000,E1 112.823} C_DIS
LIN {X 0.197,Y -689.594,Z 1285.426,A 0.000,B 0.000,C 90.000,E1 112.717} C_DIS
LIN {X -0.014,Y -683.177,Z 1285.424,A 0.000,B 0.000,C 90.000,E1 112.386} C_DIS
LIN {X -0.041,Y -679.393,Z 1285.424,A 0.000,B 0.000,C 90.000,E1 112.259} C_DIS
LIN {X 0.183,Y -670.080,Z 1285.423,A 0.000,B 0.000,C 90.000,E1 112.078} C_DIS
LIN {X -0.125,Y -664.196,Z 1285.423,A 0.000,B 0.000,C 90.000,E1 112.078} C_DIS
LIN {X -0.177,Y -641.355,Z 1285.423,A 0.000,B 0.000,C 90.000,E1 112.078} C_DIS
LIN {X 0.052,Y -639.442,Z 1285.422,A 0.000,B 0.000,C 90.000,E1 112.025} C_DIS
LIN {X -0.091,Y -637.332,Z 1285.422,A 0.000,B 0.000,C 90.000,E1 111.972} C_DIS
LIN {X -0.126,Y -637.305,Z 1285.422,A 0.000,B 0.000,C 90.000,E1 111.972} C_DIS
LIN {X 0.176,Y -637.825,Z 1285.421,A 0.000,B 0.000,C 90.000,E1 111.791} C_DIS
LIN {X 0.198,Y -638.414,Z 1285.421,A 0.000,B 0.000,C 90.000,E1 111.663} C_DIS
LIN {X 0.201,Y -640.872,Z 1285.418,A 0.000,B 0.000,C 90.000,E1 111.280} C_DIS
LIN {X 0.002,Y -646.423,Z 1285.414,A 0.000,B 0.000,C 90.000,E1 110.556} C_DIS
LIN {X -0.087,Y -649.938,Z 1285.411,A 0.000,B 0.000,C 90.000,E1 110.066} C_DIS
LIN {X -0.115,Y -653.778,Z 1285.408,A 0.000,B 0.000,C 90.000,E1 109.450} C_DIS
LIN {X -0.117,Y -657.113,Z 1285.405,A 0.000,B 0.000,C 90.000,E1 108.833} C_DIS
LIN {X 0.365,Y -660.647,Z 1285.401,A 0.000,B 0.000,C 90.000,E1 108.055} C_DIS
LIN {X 0.057,Y -663.872,Z 1285.396,A 0.000,B 0.000,C 90.000,E1 107.347} C_DIS
LIN {X 0.068,Y -665.803,Z 1285.394,A 0.000,B 0.000,C 90.000,E1 106.858} C_DIS
LIN {X 0.004,Y -668.325,Z 1285.390,A 0.000,B 0.000,C 90.000,E1 106.134} C_DIS
LIN {X -0.223,Y -670.443,Z 1285.386,A 0.000,B 0.000,C 90.000,E1 105.426} C_DIS
LIN {X 0.163,Y -672.645,Z 1285.380,A 0.000,B 0.000,C 90.000,E1 104.426} C_DIS
LIN {X -0.013,Y -673.849,Z 1285.376,A 0.000,B 0.000,C 90.000,E1 103.716} C_DIS
LIN {X -0.179,Y -674.607,Z 1285.372,A 0.000,B 0.000,C 90.000,E1 103.008} C_DIS
LIN {X -0.287,Y -674.967,Z 1285.370,A 0.000,B 0.000,C 90.000,E1 102.535} C_DIS
LIN {X 0.265,Y -675.110,Z 1285.367,A 0.000,B 0.000,C 90.000,E1 102.007} C_DIS
LIN {X 0.156,Y -675.080,Z 1285.364,A 0.000,B 0.000,C 90.000,E1 101.535} C_DIS
LIN {X -0.141,Y -674.557,Z 1285.360,A 0.000,B 0.000,C 90.000,E1 100.838} C_DIS
LIN {X -0.259,Y -674.049,Z 1285.358,A 0.000,B 0.000,C 90.000,E1 100.366} C_DIS
LIN {X 0.163,Y -673.286,Z 1285.355,A 0.000,B 0.000,C 90.000,E1 99.849} C_DIS
LIN {X 0.031,Y -672.298,Z 1285.352,A 0.000,B 0.000,C 90.000,E1 99.378} C_DIS
LIN {X -0.216,Y -670.964,Z 1285.349,A 0.000,B 0.000,C 90.000,E1 98.916} C_DIS
LIN {X 0.193,Y -669.285,Z 1285.347,A 0.000,B 0.000,C 90.000,E1 98.398} C_DIS
LIN {X 0.112,Y -668.367,Z 1285.345,A 0.000,B 0.000,C 90.000,E1 98.163} C_DIS
LIN {X -0.155,Y -666.251,Z 1285.343,A 0.000,B 0.000,C 90.000,E1 97.701} C_DIS
LIN {X 0.133,Y -663.154,Z 1285.339,A 0.000,B 0.000,C 90.000,E1 97.068} C_DIS
LIN {X -0.164,Y -660.371,Z 1285.337,A 0.000,B 0.000,C 90.000,E1 96.606} C_DIS
LIN {X 0.144,Y -656.317,Z 1285.333,A 0.000,B 0.000,C 90.000,E1 95.967} C_DIS
LIN {X -0.264,Y -652.771,Z 1285.331,A 0.000,B 0.000,C 90.000,E1 95.511} C_DIS
LIN {X 0.020,Y -648.930,Z 1285.328,A 0.000,B 0.000,C 90.000,E1 94.992} C_DIS
LIN {X 0.158,Y -643.551,Z 1285.324,A 0.000,B 0.000,C 90.000,E1 94.359} C_DIS
LIN {X 0.249,Y -637.633,Z 1285.321,A 0.000,B 0.000,C 90.000,E1 93.726} C_DIS
LIN {X -0.061,Y -632.777,Z 1285.318,A 0.000,B 0.000,C 90.000,E1 93.269} C_DIS
LIN {X 0.277,Y -626.326,Z 1285.315,A 0.000,B 0.000,C 90.000,E1 92.636} C_DIS
LIN {X 0.116,Y -620.974,Z 1285.312,A 0.000,B 0.000,C 90.000,E1 92.178} C_DIS
LIN {X 0.124,Y -615.454,Z 1285.310,A 0.000,B 0.000,C 90.000,E1 91.718} C_DIS
LIN {X -0.243,Y -609.634,Z 1285.307,A 0.000,B 0.000,C 90.000,E1 91.318} C_DIS
LIN {X -0.179,Y -601.867,Z 1285.304,A 0.000,B 0.000,C 90.000,E1 90.802} C_DIS
LIN {X 0.093,Y -595.335,Z 1285.302,A 0.000,B 0.000,C 90.000,E1 90.401} C_DIS
LIN {X 0.097,Y -588.325,Z 1285.300,A 0.000,B 0.000,C 90.000,E1 90.057} C_DIS
LIN {X 0.041,Y -581.034,Z 1285.299,A 0.000,B 0.000,C 90.000,E1 89.771} C_DIS
LIN {X -0.219,Y -575.954,Z 1285.298,A 0.000,B 0.000,C 90.000,E1 89.599} C_DIS
LIN {X -0.264,Y -572.149,Z 1285.297,A 0.000,B 0.000,C 90.000,E1 89.427} C_DIS
LIN {X 0.260,Y -572.066,Z 1285.297,A 0.000,B 0.000,C 90.000,E1 89.370} C_DIS
LIN {X 0.225,Y -569.658,Z 1285.295,A 0.000,B 0.000,C 90.000,E1 89.083} C_DIS
LIN {X 0.183,Y -569.629,Z 1285.295,A 0.000,B 0.000,C 90.000,E1 89.083} C_DIS
LIN {X -0.207,Y -569.337,Z 1285.294,A 0.000,B 0.000,C 90.000,E1 88.969} C_DIS
LIN {X 0.142,Y -569.215,Z 1285.293,A 0.000,B 0.000,C 90.000,E1 88.797} C_DIS
LIN {X 0.137,Y -570.093,Z 1285.285,A 0.000,B 0.000,C 90.000,E1 87.249} C_DIS
LIN {X 0.129,Y -572.071,Z 1285.273,A 0.000,B 0.000,C 90.000,E1 85.065} C_DIS
LIN {X -0.079,Y -573.833,Z 1285.264,A 0.000,B 0.000,C 90.000,E1 83.451} C_DIS
LIN {X -0.055,Y -576.044,Z 1285.253,A 0.000,B 0.000,C 90.000,E1 81.546} C_DIS
LIN {X 0.122,Y -577.358,Z 1285.247,A 0.000,B 0.000,C 90.000,E1 80.443} C_DIS
LIN {X -0.257,Y -578.512,Z 1285.241,A 0.000,B 0.000,C 90.000,E1 79.398} C_DIS
LIN {X 0.280,Y -579.743,Z 1285.234,A 0.000,B 0.000,C 90.000,E1 77.993} C_DIS
LIN {X 0.047,Y -580.704,Z 1285.228,A 0.000,B 0.000,C 90.000,E1 76.937} C_DIS
END
